DATA_BLOCK "DB_NcVarSelect_MA_POS_LIMIT_MINUS2"   // DB67
{ S7_Optimized_Access := 'TRUE' }
// stored: MemoryReserve 100
   VAR
      "$MA_POS_LIMIT_MINUS2_Axis01_X" { S7_SetPoint := 'True'} : "LBP_typeNCVariableTokenLReal";
      "$MA_POS_LIMIT_MINUS2_Axis02_Y" { S7_SetPoint := 'True'} : "LBP_typeNCVariableTokenLReal";
      "$MA_POS_LIMIT_MINUS2_Axis03_ZM" { S7_SetPoint := 'True'} : "LBP_typeNCVariableTokenLReal";
      "$MA_POS_LIMIT_MINUS2_Axis04_B" { S7_SetPoint := 'True'} : "LBP_typeNCVariableTokenLReal";
      "$MA_POS_LIMIT_MINUS2_Axis05_U1" { S7_SetPoint := 'True'} : "LBP_typeNCVariableTokenLReal";
      "$MA_POS_LIMIT_MINUS2_Axis06_U2" { S7_SetPoint := 'True'} : "LBP_typeNCVariableTokenLReal";
      "$MA_POS_LIMIT_MINUS2_Axis07_V" { S7_SetPoint := 'True'} : "LBP_typeNCVariableTokenLReal";
      "$MA_POS_LIMIT_MINUS2_Axis08_W" { S7_SetPoint := 'True'} : "LBP_typeNCVariableTokenLReal";
      "$MA_POS_LIMIT_MINUS2_Axis09_ZL" { S7_SetPoint := 'True'} : "LBP_typeNCVariableTokenLReal";
   END_VAR
BEGIN
   "$MA_POS_LIMIT_MINUS2_Axis01_X".token.syntaxId := 16#82;
   "$MA_POS_LIMIT_MINUS2_Axis01_X".token.areaAndUnit := 16#61;
   "$MA_POS_LIMIT_MINUS2_Axis01_X".token.column := 16#8D18;
   "$MA_POS_LIMIT_MINUS2_Axis01_X".token.row := 16#1;
   "$MA_POS_LIMIT_MINUS2_Axis01_X".token.blockType := 16#1A;
   "$MA_POS_LIMIT_MINUS2_Axis01_X".token.numberOfRows := 16#1;
   "$MA_POS_LIMIT_MINUS2_Axis01_X".token.dataTypeCode := 16#F;
   "$MA_POS_LIMIT_MINUS2_Axis01_X".token.length := 16#8;
   "$MA_POS_LIMIT_MINUS2_Axis02_Y".token.syntaxId := 16#82;
   "$MA_POS_LIMIT_MINUS2_Axis02_Y".token.areaAndUnit := 16#62;
   "$MA_POS_LIMIT_MINUS2_Axis02_Y".token.column := 16#8D18;
   "$MA_POS_LIMIT_MINUS2_Axis02_Y".token.row := 16#1;
   "$MA_POS_LIMIT_MINUS2_Axis02_Y".token.blockType := 16#1A;
   "$MA_POS_LIMIT_MINUS2_Axis02_Y".token.numberOfRows := 16#1;
   "$MA_POS_LIMIT_MINUS2_Axis02_Y".token.dataTypeCode := 16#F;
   "$MA_POS_LIMIT_MINUS2_Axis02_Y".token.length := 16#8;
   "$MA_POS_LIMIT_MINUS2_Axis03_ZM".token.syntaxId := 16#82;
   "$MA_POS_LIMIT_MINUS2_Axis03_ZM".token.areaAndUnit := 16#63;
   "$MA_POS_LIMIT_MINUS2_Axis03_ZM".token.column := 16#8D18;
   "$MA_POS_LIMIT_MINUS2_Axis03_ZM".token.row := 16#1;
   "$MA_POS_LIMIT_MINUS2_Axis03_ZM".token.blockType := 16#1A;
   "$MA_POS_LIMIT_MINUS2_Axis03_ZM".token.numberOfRows := 16#1;
   "$MA_POS_LIMIT_MINUS2_Axis03_ZM".token.dataTypeCode := 16#F;
   "$MA_POS_LIMIT_MINUS2_Axis03_ZM".token.length := 16#8;
   "$MA_POS_LIMIT_MINUS2_Axis04_B".token.syntaxId := 16#82;
   "$MA_POS_LIMIT_MINUS2_Axis04_B".token.areaAndUnit := 16#64;
   "$MA_POS_LIMIT_MINUS2_Axis04_B".token.column := 16#8D18;
   "$MA_POS_LIMIT_MINUS2_Axis04_B".token.row := 16#1;
   "$MA_POS_LIMIT_MINUS2_Axis04_B".token.blockType := 16#1A;
   "$MA_POS_LIMIT_MINUS2_Axis04_B".token.numberOfRows := 16#1;
   "$MA_POS_LIMIT_MINUS2_Axis04_B".token.dataTypeCode := 16#F;
   "$MA_POS_LIMIT_MINUS2_Axis04_B".token.length := 16#8;
   "$MA_POS_LIMIT_MINUS2_Axis05_U1".token.syntaxId := 16#82;
   "$MA_POS_LIMIT_MINUS2_Axis05_U1".token.areaAndUnit := 16#65;
   "$MA_POS_LIMIT_MINUS2_Axis05_U1".token.column := 16#8D18;
   "$MA_POS_LIMIT_MINUS2_Axis05_U1".token.row := 16#1;
   "$MA_POS_LIMIT_MINUS2_Axis05_U1".token.blockType := 16#1A;
   "$MA_POS_LIMIT_MINUS2_Axis05_U1".token.numberOfRows := 16#1;
   "$MA_POS_LIMIT_MINUS2_Axis05_U1".token.dataTypeCode := 16#F;
   "$MA_POS_LIMIT_MINUS2_Axis05_U1".token.length := 16#8;
   "$MA_POS_LIMIT_MINUS2_Axis06_U2".token.syntaxId := 16#82;
   "$MA_POS_LIMIT_MINUS2_Axis06_U2".token.areaAndUnit := 16#66;
   "$MA_POS_LIMIT_MINUS2_Axis06_U2".token.column := 16#8D18;
   "$MA_POS_LIMIT_MINUS2_Axis06_U2".token.row := 16#1;
   "$MA_POS_LIMIT_MINUS2_Axis06_U2".token.blockType := 16#1A;
   "$MA_POS_LIMIT_MINUS2_Axis06_U2".token.numberOfRows := 16#1;
   "$MA_POS_LIMIT_MINUS2_Axis06_U2".token.dataTypeCode := 16#F;
   "$MA_POS_LIMIT_MINUS2_Axis06_U2".token.length := 16#8;
   "$MA_POS_LIMIT_MINUS2_Axis07_V".token.syntaxId := 16#82;
   "$MA_POS_LIMIT_MINUS2_Axis07_V".token.areaAndUnit := 16#67;
   "$MA_POS_LIMIT_MINUS2_Axis07_V".token.column := 16#8D18;
   "$MA_POS_LIMIT_MINUS2_Axis07_V".token.row := 16#1;
   "$MA_POS_LIMIT_MINUS2_Axis07_V".token.blockType := 16#1A;
   "$MA_POS_LIMIT_MINUS2_Axis07_V".token.numberOfRows := 16#1;
   "$MA_POS_LIMIT_MINUS2_Axis07_V".token.dataTypeCode := 16#F;
   "$MA_POS_LIMIT_MINUS2_Axis07_V".token.length := 16#8;
   "$MA_POS_LIMIT_MINUS2_Axis08_W".token.syntaxId := 16#82;
   "$MA_POS_LIMIT_MINUS2_Axis08_W".token.areaAndUnit := 16#68;
   "$MA_POS_LIMIT_MINUS2_Axis08_W".token.column := 16#8D18;
   "$MA_POS_LIMIT_MINUS2_Axis08_W".token.row := 16#1;
   "$MA_POS_LIMIT_MINUS2_Axis08_W".token.blockType := 16#1A;
   "$MA_POS_LIMIT_MINUS2_Axis08_W".token.numberOfRows := 16#1;
   "$MA_POS_LIMIT_MINUS2_Axis08_W".token.dataTypeCode := 16#F;
   "$MA_POS_LIMIT_MINUS2_Axis08_W".token.length := 16#8;
   "$MA_POS_LIMIT_MINUS2_Axis09_ZL".token.syntaxId := 16#82;
   "$MA_POS_LIMIT_MINUS2_Axis09_ZL".token.areaAndUnit := 16#69;
   "$MA_POS_LIMIT_MINUS2_Axis09_ZL".token.column := 16#8D18;
   "$MA_POS_LIMIT_MINUS2_Axis09_ZL".token.row := 16#1;
   "$MA_POS_LIMIT_MINUS2_Axis09_ZL".token.blockType := 16#1A;
   "$MA_POS_LIMIT_MINUS2_Axis09_ZL".token.numberOfRows := 16#1;
   "$MA_POS_LIMIT_MINUS2_Axis09_ZL".token.dataTypeCode := 16#F;
   "$MA_POS_LIMIT_MINUS2_Axis09_ZL".token.length := 16#8;
END_DATA_BLOCK

DATA_BLOCK "DB_NcVarSelect_MA_POS_LIMIT_PLUS"   // DB68
{ S7_Optimized_Access := 'TRUE' }
// stored: MemoryReserve 100
   VAR
      "$MA_POS_LIMIT_PLUS_Axis01_X" { S7_SetPoint := 'True'} : SINU_typeNcVarTokenLReal;
      "$MA_POS_LIMIT_PLUS_Axis02_Y" { S7_SetPoint := 'True'} : SINU_typeNcVarTokenLReal;
      "$MA_POS_LIMIT_PLUS_Axis03_ZM" { S7_SetPoint := 'True'} : SINU_typeNcVarTokenLReal;
      "$MA_POS_LIMIT_PLUS_Axis04_B" { S7_SetPoint := 'True'} : SINU_typeNcVarTokenLReal;
      "$MA_POS_LIMIT_PLUS_Axis05_U1" { S7_SetPoint := 'True'} : SINU_typeNcVarTokenLReal;
      "$MA_POS_LIMIT_PLUS_Axis06_U2" { S7_SetPoint := 'True'} : SINU_typeNcVarTokenLReal;
      "$MA_POS_LIMIT_PLUS_Axis07_V" { S7_SetPoint := 'True'} : SINU_typeNcVarTokenLReal;
      "$MA_POS_LIMIT_PLUS_Axis08_W" { S7_SetPoint := 'True'} : SINU_typeNcVarTokenLReal;
      "$MA_POS_LIMIT_PLUS_Axis09_ZL" { S7_SetPoint := 'True'} : SINU_typeNcVarTokenLReal;
   END_VAR
BEGIN
   "$MA_POS_LIMIT_PLUS_Axis01_X".token.syntaxId := 16#82;
   "$MA_POS_LIMIT_PLUS_Axis01_X".token.areaAndUnit := 16#61;
   "$MA_POS_LIMIT_PLUS_Axis01_X".token.column := 16#8D0E;
   "$MA_POS_LIMIT_PLUS_Axis01_X".token.row := 16#1;
   "$MA_POS_LIMIT_PLUS_Axis01_X".token.blockType := 16#1A;
   "$MA_POS_LIMIT_PLUS_Axis01_X".token.rowCount := 16#1;
   "$MA_POS_LIMIT_PLUS_Axis01_X".token.dataType := 16#F;
   "$MA_POS_LIMIT_PLUS_Axis01_X".token.length := 16#8;
   "$MA_POS_LIMIT_PLUS_Axis02_Y".token.syntaxId := 16#82;
   "$MA_POS_LIMIT_PLUS_Axis02_Y".token.areaAndUnit := 16#62;
   "$MA_POS_LIMIT_PLUS_Axis02_Y".token.column := 16#8D0E;
   "$MA_POS_LIMIT_PLUS_Axis02_Y".token.row := 16#1;
   "$MA_POS_LIMIT_PLUS_Axis02_Y".token.blockType := 16#1A;
   "$MA_POS_LIMIT_PLUS_Axis02_Y".token.rowCount := 16#1;
   "$MA_POS_LIMIT_PLUS_Axis02_Y".token.dataType := 16#F;
   "$MA_POS_LIMIT_PLUS_Axis02_Y".token.length := 16#8;
   "$MA_POS_LIMIT_PLUS_Axis03_ZM".token.syntaxId := 16#82;
   "$MA_POS_LIMIT_PLUS_Axis03_ZM".token.areaAndUnit := 16#63;
   "$MA_POS_LIMIT_PLUS_Axis03_ZM".token.column := 16#8D0E;
   "$MA_POS_LIMIT_PLUS_Axis03_ZM".token.row := 16#1;
   "$MA_POS_LIMIT_PLUS_Axis03_ZM".token.blockType := 16#1A;
   "$MA_POS_LIMIT_PLUS_Axis03_ZM".token.rowCount := 16#1;
   "$MA_POS_LIMIT_PLUS_Axis03_ZM".token.dataType := 16#F;
   "$MA_POS_LIMIT_PLUS_Axis03_ZM".token.length := 16#8;
   "$MA_POS_LIMIT_PLUS_Axis04_B".token.syntaxId := 16#82;
   "$MA_POS_LIMIT_PLUS_Axis04_B".token.areaAndUnit := 16#64;
   "$MA_POS_LIMIT_PLUS_Axis04_B".token.column := 16#8D0E;
   "$MA_POS_LIMIT_PLUS_Axis04_B".token.row := 16#1;
   "$MA_POS_LIMIT_PLUS_Axis04_B".token.blockType := 16#1A;
   "$MA_POS_LIMIT_PLUS_Axis04_B".token.rowCount := 16#1;
   "$MA_POS_LIMIT_PLUS_Axis04_B".token.dataType := 16#F;
   "$MA_POS_LIMIT_PLUS_Axis04_B".token.length := 16#8;
   "$MA_POS_LIMIT_PLUS_Axis05_U1".token.syntaxId := 16#82;
   "$MA_POS_LIMIT_PLUS_Axis05_U1".token.areaAndUnit := 16#65;
   "$MA_POS_LIMIT_PLUS_Axis05_U1".token.column := 16#8D0E;
   "$MA_POS_LIMIT_PLUS_Axis05_U1".token.row := 16#1;
   "$MA_POS_LIMIT_PLUS_Axis05_U1".token.blockType := 16#1A;
   "$MA_POS_LIMIT_PLUS_Axis05_U1".token.rowCount := 16#1;
   "$MA_POS_LIMIT_PLUS_Axis05_U1".token.dataType := 16#F;
   "$MA_POS_LIMIT_PLUS_Axis05_U1".token.length := 16#8;
   "$MA_POS_LIMIT_PLUS_Axis06_U2".token.syntaxId := 16#82;
   "$MA_POS_LIMIT_PLUS_Axis06_U2".token.areaAndUnit := 16#66;
   "$MA_POS_LIMIT_PLUS_Axis06_U2".token.column := 16#8D0E;
   "$MA_POS_LIMIT_PLUS_Axis06_U2".token.row := 16#1;
   "$MA_POS_LIMIT_PLUS_Axis06_U2".token.blockType := 16#1A;
   "$MA_POS_LIMIT_PLUS_Axis06_U2".token.rowCount := 16#1;
   "$MA_POS_LIMIT_PLUS_Axis06_U2".token.dataType := 16#F;
   "$MA_POS_LIMIT_PLUS_Axis06_U2".token.length := 16#8;
   "$MA_POS_LIMIT_PLUS_Axis07_V".token.syntaxId := 16#82;
   "$MA_POS_LIMIT_PLUS_Axis07_V".token.areaAndUnit := 16#67;
   "$MA_POS_LIMIT_PLUS_Axis07_V".token.column := 16#8D0E;
   "$MA_POS_LIMIT_PLUS_Axis07_V".token.row := 16#1;
   "$MA_POS_LIMIT_PLUS_Axis07_V".token.blockType := 16#1A;
   "$MA_POS_LIMIT_PLUS_Axis07_V".token.rowCount := 16#1;
   "$MA_POS_LIMIT_PLUS_Axis07_V".token.dataType := 16#F;
   "$MA_POS_LIMIT_PLUS_Axis07_V".token.length := 16#8;
   "$MA_POS_LIMIT_PLUS_Axis08_W".token.syntaxId := 16#82;
   "$MA_POS_LIMIT_PLUS_Axis08_W".token.areaAndUnit := 16#68;
   "$MA_POS_LIMIT_PLUS_Axis08_W".token.column := 16#8D0E;
   "$MA_POS_LIMIT_PLUS_Axis08_W".token.row := 16#1;
   "$MA_POS_LIMIT_PLUS_Axis08_W".token.blockType := 16#1A;
   "$MA_POS_LIMIT_PLUS_Axis08_W".token.rowCount := 16#1;
   "$MA_POS_LIMIT_PLUS_Axis08_W".token.dataType := 16#F;
   "$MA_POS_LIMIT_PLUS_Axis08_W".token.length := 16#8;
   "$MA_POS_LIMIT_PLUS_Axis09_ZL".token.syntaxId := 16#82;
   "$MA_POS_LIMIT_PLUS_Axis09_ZL".token.areaAndUnit := 16#69;
   "$MA_POS_LIMIT_PLUS_Axis09_ZL".token.column := 16#8D0E;
   "$MA_POS_LIMIT_PLUS_Axis09_ZL".token.row := 16#1;
   "$MA_POS_LIMIT_PLUS_Axis09_ZL".token.blockType := 16#1A;
   "$MA_POS_LIMIT_PLUS_Axis09_ZL".token.rowCount := 16#1;
   "$MA_POS_LIMIT_PLUS_Axis09_ZL".token.dataType := 16#F;
   "$MA_POS_LIMIT_PLUS_Axis09_ZL".token.length := 16#8;
END_DATA_BLOCK

DATA_BLOCK "DB_NcVarSelect_MA_POS_LIMIT_PLUS2"   // DB69
{ S7_Optimized_Access := 'TRUE' }
// stored: MemoryReserve 100
   VAR
      "$MA_POS_LIMIT_PLUS2_Axis01_X" { S7_SetPoint := 'True'} : "LBP_typeNCVariableTokenLReal";
      "$MA_POS_LIMIT_PLUS2_Axis02_Y" { S7_SetPoint := 'True'} : "LBP_typeNCVariableTokenLReal";
      "$MA_POS_LIMIT_PLUS2_Axis03_ZM" { S7_SetPoint := 'True'} : "LBP_typeNCVariableTokenLReal";
      "$MA_POS_LIMIT_PLUS2_Axis04_B" { S7_SetPoint := 'True'} : "LBP_typeNCVariableTokenLReal";
      "$MA_POS_LIMIT_PLUS2_Axis05_U1" { S7_SetPoint := 'True'} : "LBP_typeNCVariableTokenLReal";
      "$MA_POS_LIMIT_PLUS2_Axis06_U2" { S7_SetPoint := 'True'} : "LBP_typeNCVariableTokenLReal";
      "$MA_POS_LIMIT_PLUS2_Axis07_V" { S7_SetPoint := 'True'} : "LBP_typeNCVariableTokenLReal";
      "$MA_POS_LIMIT_PLUS2_Axis08_W" { S7_SetPoint := 'True'} : "LBP_typeNCVariableTokenLReal";
      "$MA_POS_LIMIT_PLUS2_Axis09_ZL" { S7_SetPoint := 'True'} : "LBP_typeNCVariableTokenLReal";
   END_VAR
BEGIN
   "$MA_POS_LIMIT_PLUS2_Axis01_X".token.syntaxId := 16#82;
   "$MA_POS_LIMIT_PLUS2_Axis01_X".token.areaAndUnit := 16#61;
   "$MA_POS_LIMIT_PLUS2_Axis01_X".token.column := 16#8D22;
   "$MA_POS_LIMIT_PLUS2_Axis01_X".token.row := 16#1;
   "$MA_POS_LIMIT_PLUS2_Axis01_X".token.blockType := 16#1A;
   "$MA_POS_LIMIT_PLUS2_Axis01_X".token.numberOfRows := 16#1;
   "$MA_POS_LIMIT_PLUS2_Axis01_X".token.dataTypeCode := 16#F;
   "$MA_POS_LIMIT_PLUS2_Axis01_X".token.length := 16#8;
   "$MA_POS_LIMIT_PLUS2_Axis02_Y".token.syntaxId := 16#82;
   "$MA_POS_LIMIT_PLUS2_Axis02_Y".token.areaAndUnit := 16#62;
   "$MA_POS_LIMIT_PLUS2_Axis02_Y".token.column := 16#8D22;
   "$MA_POS_LIMIT_PLUS2_Axis02_Y".token.row := 16#1;
   "$MA_POS_LIMIT_PLUS2_Axis02_Y".token.blockType := 16#1A;
   "$MA_POS_LIMIT_PLUS2_Axis02_Y".token.numberOfRows := 16#1;
   "$MA_POS_LIMIT_PLUS2_Axis02_Y".token.dataTypeCode := 16#F;
   "$MA_POS_LIMIT_PLUS2_Axis02_Y".token.length := 16#8;
   "$MA_POS_LIMIT_PLUS2_Axis03_ZM".token.syntaxId := 16#82;
   "$MA_POS_LIMIT_PLUS2_Axis03_ZM".token.areaAndUnit := 16#63;
   "$MA_POS_LIMIT_PLUS2_Axis03_ZM".token.column := 16#8D22;
   "$MA_POS_LIMIT_PLUS2_Axis03_ZM".token.row := 16#1;
   "$MA_POS_LIMIT_PLUS2_Axis03_ZM".token.blockType := 16#1A;
   "$MA_POS_LIMIT_PLUS2_Axis03_ZM".token.numberOfRows := 16#1;
   "$MA_POS_LIMIT_PLUS2_Axis03_ZM".token.dataTypeCode := 16#F;
   "$MA_POS_LIMIT_PLUS2_Axis03_ZM".token.length := 16#8;
   "$MA_POS_LIMIT_PLUS2_Axis04_B".token.syntaxId := 16#82;
   "$MA_POS_LIMIT_PLUS2_Axis04_B".token.areaAndUnit := 16#64;
   "$MA_POS_LIMIT_PLUS2_Axis04_B".token.column := 16#8D22;
   "$MA_POS_LIMIT_PLUS2_Axis04_B".token.row := 16#1;
   "$MA_POS_LIMIT_PLUS2_Axis04_B".token.blockType := 16#1A;
   "$MA_POS_LIMIT_PLUS2_Axis04_B".token.numberOfRows := 16#1;
   "$MA_POS_LIMIT_PLUS2_Axis04_B".token.dataTypeCode := 16#F;
   "$MA_POS_LIMIT_PLUS2_Axis04_B".token.length := 16#8;
   "$MA_POS_LIMIT_PLUS2_Axis05_U1".token.syntaxId := 16#82;
   "$MA_POS_LIMIT_PLUS2_Axis05_U1".token.areaAndUnit := 16#65;
   "$MA_POS_LIMIT_PLUS2_Axis05_U1".token.column := 16#8D22;
   "$MA_POS_LIMIT_PLUS2_Axis05_U1".token.row := 16#1;
   "$MA_POS_LIMIT_PLUS2_Axis05_U1".token.blockType := 16#1A;
   "$MA_POS_LIMIT_PLUS2_Axis05_U1".token.numberOfRows := 16#1;
   "$MA_POS_LIMIT_PLUS2_Axis05_U1".token.dataTypeCode := 16#F;
   "$MA_POS_LIMIT_PLUS2_Axis05_U1".token.length := 16#8;
   "$MA_POS_LIMIT_PLUS2_Axis06_U2".token.syntaxId := 16#82;
   "$MA_POS_LIMIT_PLUS2_Axis06_U2".token.areaAndUnit := 16#66;
   "$MA_POS_LIMIT_PLUS2_Axis06_U2".token.column := 16#8D22;
   "$MA_POS_LIMIT_PLUS2_Axis06_U2".token.row := 16#1;
   "$MA_POS_LIMIT_PLUS2_Axis06_U2".token.blockType := 16#1A;
   "$MA_POS_LIMIT_PLUS2_Axis06_U2".token.numberOfRows := 16#1;
   "$MA_POS_LIMIT_PLUS2_Axis06_U2".token.dataTypeCode := 16#F;
   "$MA_POS_LIMIT_PLUS2_Axis06_U2".token.length := 16#8;
   "$MA_POS_LIMIT_PLUS2_Axis07_V".token.syntaxId := 16#82;
   "$MA_POS_LIMIT_PLUS2_Axis07_V".token.areaAndUnit := 16#67;
   "$MA_POS_LIMIT_PLUS2_Axis07_V".token.column := 16#8D22;
   "$MA_POS_LIMIT_PLUS2_Axis07_V".token.row := 16#1;
   "$MA_POS_LIMIT_PLUS2_Axis07_V".token.blockType := 16#1A;
   "$MA_POS_LIMIT_PLUS2_Axis07_V".token.numberOfRows := 16#1;
   "$MA_POS_LIMIT_PLUS2_Axis07_V".token.dataTypeCode := 16#F;
   "$MA_POS_LIMIT_PLUS2_Axis07_V".token.length := 16#8;
   "$MA_POS_LIMIT_PLUS2_Axis08_W".token.syntaxId := 16#82;
   "$MA_POS_LIMIT_PLUS2_Axis08_W".token.areaAndUnit := 16#68;
   "$MA_POS_LIMIT_PLUS2_Axis08_W".token.column := 16#8D22;
   "$MA_POS_LIMIT_PLUS2_Axis08_W".token.row := 16#1;
   "$MA_POS_LIMIT_PLUS2_Axis08_W".token.blockType := 16#1A;
   "$MA_POS_LIMIT_PLUS2_Axis08_W".token.numberOfRows := 16#1;
   "$MA_POS_LIMIT_PLUS2_Axis08_W".token.dataTypeCode := 16#F;
   "$MA_POS_LIMIT_PLUS2_Axis08_W".token.length := 16#8;
   "$MA_POS_LIMIT_PLUS2_Axis09_ZL".token.syntaxId := 16#82;
   "$MA_POS_LIMIT_PLUS2_Axis09_ZL".token.areaAndUnit := 16#69;
   "$MA_POS_LIMIT_PLUS2_Axis09_ZL".token.column := 16#8D22;
   "$MA_POS_LIMIT_PLUS2_Axis09_ZL".token.row := 16#1;
   "$MA_POS_LIMIT_PLUS2_Axis09_ZL".token.blockType := 16#1A;
   "$MA_POS_LIMIT_PLUS2_Axis09_ZL".token.numberOfRows := 16#1;
   "$MA_POS_LIMIT_PLUS2_Axis09_ZL".token.dataTypeCode := 16#F;
   "$MA_POS_LIMIT_PLUS2_Axis09_ZL".token.length := 16#8;
END_DATA_BLOCK

DATA_BLOCK "DB_NcVarSelect_M_MAX_AX_VELO"   // DB98
{ S7_Optimized_Access := 'TRUE' }
// stored: MemoryReserve 100
   VAR
      "$MA_JOG_VELO_Axis01_X" { S7_SetPoint := 'True'} : "LBP_typeNCVariableTokenLReal";
      "$MA_JOG_VELO_Axis02_Y" { S7_SetPoint := 'True'} : "LBP_typeNCVariableTokenLReal";
      "$MA_JOG_VELO_Axis03_ZM" { S7_SetPoint := 'True'} : "LBP_typeNCVariableTokenLReal";
      "$MA_JOG_VELO_Axis04_B" { S7_SetPoint := 'True'} : "LBP_typeNCVariableTokenLReal";
      "$MA_JOG_VELO_Axis05_U1" { S7_SetPoint := 'True'} : "LBP_typeNCVariableTokenLReal";
      "$MA_JOG_VELO_Axis06_U2" { S7_SetPoint := 'True'} : "LBP_typeNCVariableTokenLReal";
      "$MA_JOG_VELO_Axis07_V" { S7_SetPoint := 'True'} : "LBP_typeNCVariableTokenLReal";
      "$MA_JOG_VELO_Axis08_W" { S7_SetPoint := 'True'} : "LBP_typeNCVariableTokenLReal";
      "$MA_JOG_VELO_Axis09_ZL" { S7_SetPoint := 'True'} : "LBP_typeNCVariableTokenLReal";
   END_VAR
BEGIN
   "$MA_JOG_VELO_Axis01_X".token.syntaxId := 16#82;
   "$MA_JOG_VELO_Axis01_X".token.areaAndUnit := 16#61;
   "$MA_JOG_VELO_Axis01_X".token.column := 16#7D00;
   "$MA_JOG_VELO_Axis01_X".token.row := 16#1;
   "$MA_JOG_VELO_Axis01_X".token.blockType := 16#1A;
   "$MA_JOG_VELO_Axis01_X".token.numberOfRows := 16#1;
   "$MA_JOG_VELO_Axis01_X".token.dataTypeCode := 16#F;
   "$MA_JOG_VELO_Axis01_X".token.length := 16#8;
   "$MA_JOG_VELO_Axis02_Y".token.syntaxId := 16#82;
   "$MA_JOG_VELO_Axis02_Y".token.areaAndUnit := 16#62;
   "$MA_JOG_VELO_Axis02_Y".token.column := 16#7D00;
   "$MA_JOG_VELO_Axis02_Y".token.row := 16#1;
   "$MA_JOG_VELO_Axis02_Y".token.blockType := 16#1A;
   "$MA_JOG_VELO_Axis02_Y".token.numberOfRows := 16#1;
   "$MA_JOG_VELO_Axis02_Y".token.dataTypeCode := 16#F;
   "$MA_JOG_VELO_Axis02_Y".token.length := 16#8;
   "$MA_JOG_VELO_Axis03_ZM".token.syntaxId := 16#82;
   "$MA_JOG_VELO_Axis03_ZM".token.areaAndUnit := 16#63;
   "$MA_JOG_VELO_Axis03_ZM".token.column := 16#7D00;
   "$MA_JOG_VELO_Axis03_ZM".token.row := 16#1;
   "$MA_JOG_VELO_Axis03_ZM".token.blockType := 16#1A;
   "$MA_JOG_VELO_Axis03_ZM".token.numberOfRows := 16#1;
   "$MA_JOG_VELO_Axis03_ZM".token.dataTypeCode := 16#F;
   "$MA_JOG_VELO_Axis03_ZM".token.length := 16#8;
   "$MA_JOG_VELO_Axis04_B".token.syntaxId := 16#82;
   "$MA_JOG_VELO_Axis04_B".token.areaAndUnit := 16#64;
   "$MA_JOG_VELO_Axis04_B".token.column := 16#7D00;
   "$MA_JOG_VELO_Axis04_B".token.row := 16#1;
   "$MA_JOG_VELO_Axis04_B".token.blockType := 16#1A;
   "$MA_JOG_VELO_Axis04_B".token.numberOfRows := 16#1;
   "$MA_JOG_VELO_Axis04_B".token.dataTypeCode := 16#F;
   "$MA_JOG_VELO_Axis04_B".token.length := 16#8;
   "$MA_JOG_VELO_Axis05_U1".token.syntaxId := 16#82;
   "$MA_JOG_VELO_Axis05_U1".token.areaAndUnit := 16#65;
   "$MA_JOG_VELO_Axis05_U1".token.column := 16#7D00;
   "$MA_JOG_VELO_Axis05_U1".token.row := 16#1;
   "$MA_JOG_VELO_Axis05_U1".token.blockType := 16#1A;
   "$MA_JOG_VELO_Axis05_U1".token.numberOfRows := 16#1;
   "$MA_JOG_VELO_Axis05_U1".token.dataTypeCode := 16#F;
   "$MA_JOG_VELO_Axis05_U1".token.length := 16#8;
   "$MA_JOG_VELO_Axis06_U2".token.syntaxId := 16#82;
   "$MA_JOG_VELO_Axis06_U2".token.areaAndUnit := 16#66;
   "$MA_JOG_VELO_Axis06_U2".token.column := 16#7D00;
   "$MA_JOG_VELO_Axis06_U2".token.row := 16#1;
   "$MA_JOG_VELO_Axis06_U2".token.blockType := 16#1A;
   "$MA_JOG_VELO_Axis06_U2".token.numberOfRows := 16#1;
   "$MA_JOG_VELO_Axis06_U2".token.dataTypeCode := 16#F;
   "$MA_JOG_VELO_Axis06_U2".token.length := 16#8;
   "$MA_JOG_VELO_Axis07_V".token.syntaxId := 16#82;
   "$MA_JOG_VELO_Axis07_V".token.areaAndUnit := 16#67;
   "$MA_JOG_VELO_Axis07_V".token.column := 16#7D00;
   "$MA_JOG_VELO_Axis07_V".token.row := 16#1;
   "$MA_JOG_VELO_Axis07_V".token.blockType := 16#1A;
   "$MA_JOG_VELO_Axis07_V".token.numberOfRows := 16#1;
   "$MA_JOG_VELO_Axis07_V".token.dataTypeCode := 16#F;
   "$MA_JOG_VELO_Axis07_V".token.length := 16#8;
   "$MA_JOG_VELO_Axis08_W".token.syntaxId := 16#82;
   "$MA_JOG_VELO_Axis08_W".token.areaAndUnit := 16#68;
   "$MA_JOG_VELO_Axis08_W".token.column := 16#7D00;
   "$MA_JOG_VELO_Axis08_W".token.row := 16#1;
   "$MA_JOG_VELO_Axis08_W".token.blockType := 16#1A;
   "$MA_JOG_VELO_Axis08_W".token.numberOfRows := 16#1;
   "$MA_JOG_VELO_Axis08_W".token.dataTypeCode := 16#F;
   "$MA_JOG_VELO_Axis08_W".token.length := 16#8;
   "$MA_JOG_VELO_Axis09_ZL".token.syntaxId := 16#82;
   "$MA_JOG_VELO_Axis09_ZL".token.areaAndUnit := 16#69;
   "$MA_JOG_VELO_Axis09_ZL".token.column := 16#7D00;
   "$MA_JOG_VELO_Axis09_ZL".token.row := 16#1;
   "$MA_JOG_VELO_Axis09_ZL".token.blockType := 16#1A;
   "$MA_JOG_VELO_Axis09_ZL".token.numberOfRows := 16#1;
   "$MA_JOG_VELO_Axis09_ZL".token.dataTypeCode := 16#F;
   "$MA_JOG_VELO_Axis09_ZL".token.length := 16#8;
END_DATA_BLOCK

DATA_BLOCK "DB_AnalogInputAction"   // DB1304
TITLE = TEMPERATURE SETTINGS
{ S7_Optimized_Access := 'FALSE'; DB_Accessible_From_OPC_UA := 'FALSE' }
AUTHOR : SAN
// stored: AutoNumber false, DBAccessibleFromOPCUA false, DBAccessibleFromWebserver false
   VAR
      Laser_Power_Meter : "AnalogInAction_DT";
      Axis_B_Clamping_Part : "AnalogInAction_DT";
      Laser_Air_Pressure_Process : "AnalogInAction_DT";
      Inlet_Air_Pressure : "AnalogInAction_DT";
      Ambiant_Temperature : "AnalogInAction_DT";
      Machine_Temperature : "AnalogInAction_DT";
      Cold_Water_Temperature_Input : "AnalogInAction_DT";
      Cold_Water_Temperature_Output : "AnalogInAction_DT";
      X_Axis_Temperature_PT1000 : "AnalogInAction_DT";
      Y_Axis_Temperature_PT1000 : "AnalogInAction_DT";
      X_Axis_Temperature_PTC : "AnalogInAction_DT";
      Y_Axis_Temperature_PTC : "AnalogInAction_DT";
      Nozzle_Overpressure : "AnalogInAction_DT";
      Optical_Path_Overpressure : "AnalogInAction_DT";
      Laser_Head_Overpressure : "AnalogInAction_DT";
      ZL_Axis_Overpressure : "AnalogInAction_DT";
      XY_Axis_Overpressure : "AnalogInAction_DT";
      Left_Aspiration : "AnalogInAction_DT";
      Right_Aspiration : "AnalogInAction_DT";
      Free_IW458 : "AnalogInAction_DT";
      Clim_Temperature : "AnalogInAction_DT";
      Free_IW482 : "AnalogInAction_DT";
      Free_IW484 : "AnalogInAction_DT";
      Free_IW486 : "AnalogInAction_DT";
      Sensor_Controller_Station1 : "AnalogInAction_DT";
      Cabinet_Temperature : "AnalogInAction_DT";
      Free_IW464 : "AnalogInAction_DT";
      Free_IW466 : "AnalogInAction_DT";
   END_VAR
BEGIN
   Laser_Power_Meter.ID_Measure := 1;
   Axis_B_Clamping_Part.ID_Measure := 2;
   Laser_Air_Pressure_Process.ID_Measure := 3;
   Inlet_Air_Pressure.ID_Measure := 4;
   Ambiant_Temperature.ID_Measure := 5;
   Machine_Temperature.ID_Measure := 6;
   Cold_Water_Temperature_Input.ID_Measure := 7;
   Cold_Water_Temperature_Output.ID_Measure := 8;
   X_Axis_Temperature_PT1000.ID_Measure := 9;
   Y_Axis_Temperature_PT1000.ID_Measure := 10;
   X_Axis_Temperature_PTC.ID_Measure := 11;
   Y_Axis_Temperature_PTC.ID_Measure := 12;
   Nozzle_Overpressure.ID_Measure := 13;
   Optical_Path_Overpressure.ID_Measure := 14;
   Laser_Head_Overpressure.ID_Measure := 15;
   ZL_Axis_Overpressure.ID_Measure := 16;
   XY_Axis_Overpressure.ID_Measure := 17;
   Left_Aspiration.ID_Measure := 18;
   Right_Aspiration.ID_Measure := 19;
   Free_IW458.ID_Measure := 20;
   Clim_Temperature.ID_Measure := 21;
   Free_IW482.ID_Measure := 22;
   Free_IW484.ID_Measure := 23;
   Free_IW486.ID_Measure := 24;
   Sensor_Controller_Station1.ID_Measure := 25;
   Cabinet_Temperature.ID_Measure := 26;
   Free_IW464.ID_Measure := 27;
   Free_IW466.ID_Measure := 28;
END_DATA_BLOCK

DATA_BLOCK "DB_AnalogInputDataHMI"   // DB1303
TITLE = TEMPERATURE SETTINGS
{ S7_Optimized_Access := 'FALSE'; DB_Accessible_From_OPC_UA := 'FALSE' }
AUTHOR : SAN
// stored: AutoNumber false, DBAccessibleFromOPCUA false, DBAccessibleFromWebserver false
   VAR RETAIN
      Laser_Power_Meter : "AnalogInDataHMI_DT";
      Axis_B_Clamping_Part : "AnalogInDataHMI_DT";
      Laser_Air_Pressure_Process : "AnalogInDataHMI_DT";
      Inlet_Air_Pressure : "AnalogInDataHMI_DT";
      Ambiant_Temperature : "AnalogInDataHMI_DT";
      Machine_Temperature : "AnalogInDataHMI_DT";
      Cold_Water_Temperature_Input : "AnalogInDataHMI_DT";
      Cold_Water_Temperature_Output : "AnalogInDataHMI_DT";
      X_Axis_Temperature_PT1000 { S7_SetPoint := 'True'} : "AnalogInDataHMI_DT";
      Y_Axis_Temperature_PT1000 : "AnalogInDataHMI_DT";
      X_Axis_Temperature_PTC : "AnalogInDataHMI_DT";
      Y_Axis_Temperature_PTC : "AnalogInDataHMI_DT";
      Nozzle_Overpressure : "AnalogInDataHMI_DT";
      Optical_Path_Overpressure : "AnalogInDataHMI_DT";
      Laser_Head_Overpressure : "AnalogInDataHMI_DT";
      ZL_Axis_Overpressure : "AnalogInDataHMI_DT";
      XY_Axis_Overpressure : "AnalogInDataHMI_DT";
      Left_Aspiration : "AnalogInDataHMI_DT";
      Right_Aspiration : "AnalogInDataHMI_DT";
      Free_IW458 : "AnalogInDataHMI_DT";
      Clim_Temperature : "AnalogInDataHMI_DT";
      Free_IW482 : "AnalogInDataHMI_DT";
      Free_IW484 : "AnalogInDataHMI_DT";
      Free_IW486 : "AnalogInDataHMI_DT";
      Sensor_Controller_Station1 : "AnalogInDataHMI_DT";
      Cabinet_Temperature : "AnalogInDataHMI_DT";
      Free_IW464 : "AnalogInDataHMI_DT";
      Free_IW466 : "AnalogInDataHMI_DT";
   END_VAR
BEGIN
   Laser_Power_Meter.ID_Measure := 701;
   Axis_B_Clamping_Part.ID_Measure := 810;
   Laser_Air_Pressure_Process.ID_Measure := 511;
   Laser_Air_Pressure_Process.TargetValue := 2.0;
   Laser_Air_Pressure_Process.ThresholdAlarmMin := -0.2;
   Laser_Air_Pressure_Process.ThresholdWarningMin := -0.15;
   Laser_Air_Pressure_Process.ThresholdWarningMax := 0.15;
   Laser_Air_Pressure_Process.ThresholdAlarmMax := 0.2;
   Laser_Air_Pressure_Process.StartTime := T#5s;
   Inlet_Air_Pressure.ID_Measure := 501;
   Inlet_Air_Pressure.TargetValue := 6.0;
   Inlet_Air_Pressure.ThresholdAlarmMin := -0.5;
   Inlet_Air_Pressure.ThresholdWarningMin := -0.4;
   Inlet_Air_Pressure.ThresholdWarningMax := 0.4;
   Inlet_Air_Pressure.ThresholdAlarmMax := 0.5;
   Inlet_Air_Pressure.StartTime := T#5s;
   Ambiant_Temperature.ID_Measure := 201;
   Ambiant_Temperature.TargetValue := 25.0;
   Ambiant_Temperature.ThresholdAlarmMin := -5.0;
   Ambiant_Temperature.ThresholdWarningMin := -3.0;
   Ambiant_Temperature.ThresholdWarningMax := 3.0;
   Ambiant_Temperature.ThresholdAlarmMax := 5.0;
   Machine_Temperature.ID_Measure := 202;
   Machine_Temperature.TargetValue := 25.0;
   Machine_Temperature.ThresholdAlarmMin := -5.0;
   Machine_Temperature.ThresholdWarningMin := -3.0;
   Machine_Temperature.ThresholdWarningMax := 3.0;
   Machine_Temperature.ThresholdAlarmMax := 5.0;
   Cold_Water_Temperature_Input.ID_Measure := 301;
   Cold_Water_Temperature_Input.TargetValue := 23.0;
   Cold_Water_Temperature_Input.ThresholdAlarmMin := -3.0;
   Cold_Water_Temperature_Input.ThresholdWarningMin := -2.0;
   Cold_Water_Temperature_Input.ThresholdWarningMax := 2.0;
   Cold_Water_Temperature_Input.ThresholdAlarmMax := 3.0;
   Cold_Water_Temperature_Output.ID_Measure := 302;
   Cold_Water_Temperature_Output.TargetValue := 24.0;
   Cold_Water_Temperature_Output.ThresholdAlarmMin := -3.0;
   Cold_Water_Temperature_Output.ThresholdWarningMin := -2.0;
   Cold_Water_Temperature_Output.ThresholdWarningMax := 2.0;
   Cold_Water_Temperature_Output.ThresholdAlarmMax := 3.0;
   X_Axis_Temperature_PT1000.ID_Measure := 110;
   X_Axis_Temperature_PT1000.TargetValue := 25.0;
   X_Axis_Temperature_PT1000.ThresholdAlarmMin := -5.0;
   X_Axis_Temperature_PT1000.ThresholdWarningMin := -3.0;
   X_Axis_Temperature_PT1000.ThresholdWarningMax := 3.0;
   X_Axis_Temperature_PT1000.ThresholdAlarmMax := 5.0;
   X_Axis_Temperature_PT1000.AxFactor := 1.0;
   X_Axis_Temperature_PT1000.StartTime := T#45S;
   Y_Axis_Temperature_PT1000.ID_Measure := 120;
   Y_Axis_Temperature_PT1000.TargetValue := 25.0;
   Y_Axis_Temperature_PT1000.ThresholdAlarmMin := -5.0;
   Y_Axis_Temperature_PT1000.ThresholdWarningMin := -3.0;
   Y_Axis_Temperature_PT1000.ThresholdWarningMax := 3.0;
   Y_Axis_Temperature_PT1000.ThresholdAlarmMax := 5.0;
   X_Axis_Temperature_PTC.ID_Measure := 116;
   Y_Axis_Temperature_PTC.ID_Measure := 126;
   Nozzle_Overpressure.ID_Measure := 512;
   Nozzle_Overpressure.TargetValue := 2.0;
   Nozzle_Overpressure.ThresholdAlarmMin := -0.2;
   Nozzle_Overpressure.ThresholdWarningMin := -0.15;
   Nozzle_Overpressure.ThresholdWarningMax := 0.15;
   Nozzle_Overpressure.ThresholdAlarmMax := 0.2;
   Nozzle_Overpressure.StartTime := T#5s;
   Optical_Path_Overpressure.ID_Measure := 513;
   Optical_Path_Overpressure.TargetValue := 0.4;
   Optical_Path_Overpressure.ThresholdAlarmMin := -0.2;
   Optical_Path_Overpressure.ThresholdWarningMin := -0.19;
   Optical_Path_Overpressure.ThresholdWarningMax := 0.19;
   Optical_Path_Overpressure.ThresholdAlarmMax := 0.2;
   Optical_Path_Overpressure.StartTime := T#5s;
   Laser_Head_Overpressure.ID_Measure := 514;
   Laser_Head_Overpressure.TargetValue := 1.4;
   Laser_Head_Overpressure.ThresholdAlarmMin := -0.15;
   Laser_Head_Overpressure.ThresholdWarningMin := -0.1;
   Laser_Head_Overpressure.ThresholdWarningMax := 0.1;
   Laser_Head_Overpressure.ThresholdAlarmMax := 0.15;
   Laser_Head_Overpressure.StartTime := T#5s;
   ZL_Axis_Overpressure.ID_Measure := 520;
   ZL_Axis_Overpressure.TargetValue := 0.85;
   ZL_Axis_Overpressure.ThresholdAlarmMin := -0.2;
   ZL_Axis_Overpressure.ThresholdWarningMin := -0.15;
   ZL_Axis_Overpressure.ThresholdWarningMax := 0.15;
   ZL_Axis_Overpressure.ThresholdAlarmMax := 0.2;
   ZL_Axis_Overpressure.StartTime := T#5s;
   XY_Axis_Overpressure.ID_Measure := 530;
   XY_Axis_Overpressure.TargetValue := 0.85;
   XY_Axis_Overpressure.ThresholdAlarmMin := -0.2;
   XY_Axis_Overpressure.ThresholdWarningMin := -0.15;
   XY_Axis_Overpressure.ThresholdWarningMax := 0.15;
   XY_Axis_Overpressure.ThresholdAlarmMax := 0.2;
   XY_Axis_Overpressure.StartTime := T#5s;
   Left_Aspiration.ID_Measure := 401;
   Left_Aspiration.CurrentValue := 1.4774;
   Left_Aspiration.TargetValue := 1900.0;
   Left_Aspiration.ThresholdAlarmMin := -1000.0;
   Left_Aspiration.ThresholdWarningMin := -500.0;
   Left_Aspiration.ThresholdWarningMax := 500.0;
   Left_Aspiration.ThresholdAlarmMax := 1000.0;
   Left_Aspiration.StartTime := T#120s;
   Right_Aspiration.ID_Measure := 402;
   Right_Aspiration.CurrentValue := 1.4774;
   Right_Aspiration.TargetValue := 1900.0;
   Right_Aspiration.ThresholdAlarmMin := -1000.0;
   Right_Aspiration.ThresholdWarningMin := -500.0;
   Right_Aspiration.ThresholdWarningMax := 500.0;
   Right_Aspiration.ThresholdAlarmMax := 1000.0;
   Right_Aspiration.StartTime := T#120s;
   Free_IW458.ID_Measure := 999;
   Clim_Temperature.ID_Measure := 204;
   Free_IW482.ID_Measure := 999;
   Free_IW484.ID_Measure := 999;
   Free_IW486.ID_Measure := 999;
   Sensor_Controller_Station1.ID_Measure := 711;
   Cabinet_Temperature.ID_Measure := 203;
   Free_IW464.ID_Measure := 999;
   Free_IW466.ID_Measure := 999;
END_DATA_BLOCK

DATA_BLOCK "DB_AnalogInputDataPLC"   // DB1307
TITLE = TEMPERATURE SETTINGS
{ S7_Optimized_Access := 'FALSE'; DB_Accessible_From_OPC_UA := 'FALSE' }
AUTHOR : SAN
// stored: AutoNumber false, DBAccessibleFromOPCUA false, DBAccessibleFromWebserver false
   VAR RETAIN
      Laser_Power_Meter : "AnalogInDataPLC_DT";
      Axis_B_Clamping_Part : "AnalogInDataPLC_DT";
      Laser_Air_Pressure_Process : "AnalogInDataPLC_DT";
      Inlet_Air_Pressure : "AnalogInDataPLC_DT";
      Ambiant_Temperature : "AnalogInDataPLC_DT";
      Machine_Temperature : "AnalogInDataPLC_DT";
      Cold_Water_Temperature_Input : "AnalogInDataPLC_DT";
      Cold_Water_Temperature_Output : "AnalogInDataPLC_DT";
      X_Axis_Temperature_PT1000 : "AnalogInDataPLC_DT";
      Y_Axis_Temperature_PT1000 : "AnalogInDataPLC_DT";
      X_Axis_Temperature_PTC : "AnalogInDataPLC_DT";
      Y_Axis_Temperature_PTC : "AnalogInDataPLC_DT";
      Nozzle_Overpressure : "AnalogInDataPLC_DT";
      Optical_Path_Overpressure : "AnalogInDataPLC_DT";
      Laser_Head_Overpressure : "AnalogInDataPLC_DT";
      ZL_Axis_Overpressure : "AnalogInDataPLC_DT";
      XY_Axis_Overpressure : "AnalogInDataPLC_DT";
      Left_Aspiration : "AnalogInDataPLC_DT";
      Right_Aspiration : "AnalogInDataPLC_DT";
      Free_IW458 : "AnalogInDataPLC_DT";
      Clim_Temperature : "AnalogInDataPLC_DT";
      Free_IW482 : "AnalogInDataPLC_DT";
      Free_IW484 : "AnalogInDataPLC_DT";
      Free_IW486 : "AnalogInDataPLC_DT";
      Sensor_Controller_Station1 : "AnalogInDataPLC_DT";
      Cabinet_Temperature : "AnalogInDataPLC_DT";
      Free_IW464 : "AnalogInDataPLC_DT";
      Free_IW466 : "AnalogInDataPLC_DT";
   END_VAR
BEGIN
   Laser_Power_Meter.LimitUp := 10.0;
   Laser_Power_Meter.LimitDown := 0.0;
   Laser_Power_Meter.TypeProbe := 2;
   Axis_B_Clamping_Part.LimitUp := 27648.0;
   Axis_B_Clamping_Part.LimitDown := 0.0;
   Axis_B_Clamping_Part.TypeProbe := 2;
   Laser_Air_Pressure_Process.LimitUp := 10.0;
   Laser_Air_Pressure_Process.LimitDown := 0.0;
   Laser_Air_Pressure_Process.TypeProbe := 2;
   Laser_Air_Pressure_Process.EnableAlarmMin := True;
   Laser_Air_Pressure_Process.EnableWarningMin := True;
   Laser_Air_Pressure_Process.EnableWarningMax := True;
   Laser_Air_Pressure_Process.EnableAlarmMax := True;
   Inlet_Air_Pressure.LimitUp := 10.0;
   Inlet_Air_Pressure.LimitDown := 0.0;
   Inlet_Air_Pressure.TypeProbe := 2;
   Inlet_Air_Pressure.EnableAlarmMin := True;
   Inlet_Air_Pressure.EnableWarningMin := True;
   Inlet_Air_Pressure.EnableWarningMax := True;
   Inlet_Air_Pressure.EnableAlarmMax := True;
   Ambiant_Temperature.TypeProbe := 0;
   Ambiant_Temperature.EnableAlarmMin := True;
   Ambiant_Temperature.EnableWarningMin := True;
   Ambiant_Temperature.EnableWarningMax := True;
   Ambiant_Temperature.EnableAlarmMax := True;
   Machine_Temperature.TypeProbe := 0;
   Machine_Temperature.EnableAlarmMin := True;
   Machine_Temperature.EnableWarningMin := True;
   Machine_Temperature.EnableWarningMax := True;
   Machine_Temperature.EnableAlarmMax := True;
   Cold_Water_Temperature_Input.TypeProbe := 0;
   Cold_Water_Temperature_Input.EnableAlarmMin := True;
   Cold_Water_Temperature_Input.EnableWarningMin := True;
   Cold_Water_Temperature_Input.EnableWarningMax := True;
   Cold_Water_Temperature_Input.EnableAlarmMax := True;
   Cold_Water_Temperature_Output.TypeProbe := 0;
   Cold_Water_Temperature_Output.EnableAlarmMin := True;
   Cold_Water_Temperature_Output.EnableWarningMin := True;
   Cold_Water_Temperature_Output.EnableWarningMax := True;
   Cold_Water_Temperature_Output.EnableAlarmMax := True;
   X_Axis_Temperature_PT1000.TypeProbe := 1;
   X_Axis_Temperature_PT1000.EnableAlarmMin := True;
   X_Axis_Temperature_PT1000.EnableWarningMin := True;
   X_Axis_Temperature_PT1000.EnableWarningMax := True;
   X_Axis_Temperature_PT1000.EnableAlarmMax := True;
   Y_Axis_Temperature_PT1000.TypeProbe := 1;
   Y_Axis_Temperature_PT1000.EnableAlarmMin := True;
   Y_Axis_Temperature_PT1000.EnableWarningMin := True;
   Y_Axis_Temperature_PT1000.EnableWarningMax := True;
   Y_Axis_Temperature_PT1000.EnableAlarmMax := True;
   X_Axis_Temperature_PTC.TypeProbe := 6;
   Y_Axis_Temperature_PTC.TypeProbe := 6;
   Nozzle_Overpressure.LimitUp := 10.0;
   Nozzle_Overpressure.LimitDown := 0.0;
   Nozzle_Overpressure.TypeProbe := 2;
   Nozzle_Overpressure.EnableAlarmMin := True;
   Nozzle_Overpressure.EnableWarningMin := True;
   Nozzle_Overpressure.EnableWarningMax := True;
   Nozzle_Overpressure.EnableAlarmMax := True;
   Optical_Path_Overpressure.LimitUp := 10.0;
   Optical_Path_Overpressure.LimitDown := 0.0;
   Optical_Path_Overpressure.TypeProbe := 2;
   Optical_Path_Overpressure.EnableAlarmMin := True;
   Optical_Path_Overpressure.EnableWarningMin := True;
   Optical_Path_Overpressure.EnableWarningMax := True;
   Optical_Path_Overpressure.EnableAlarmMax := True;
   Laser_Head_Overpressure.LimitUp := 10.0;
   Laser_Head_Overpressure.LimitDown := 0.0;
   Laser_Head_Overpressure.TypeProbe := 2;
   Laser_Head_Overpressure.EnableAlarmMin := True;
   Laser_Head_Overpressure.EnableWarningMin := True;
   Laser_Head_Overpressure.EnableWarningMax := True;
   Laser_Head_Overpressure.EnableAlarmMax := True;
   ZL_Axis_Overpressure.LimitUp := 10.0;
   ZL_Axis_Overpressure.LimitDown := 0.0;
   ZL_Axis_Overpressure.TypeProbe := 2;
   ZL_Axis_Overpressure.EnableAlarmMin := True;
   ZL_Axis_Overpressure.EnableWarningMin := True;
   ZL_Axis_Overpressure.EnableWarningMax := True;
   ZL_Axis_Overpressure.EnableAlarmMax := True;
   XY_Axis_Overpressure.LimitUp := 10.0;
   XY_Axis_Overpressure.LimitDown := 0.0;
   XY_Axis_Overpressure.TypeProbe := 2;
   XY_Axis_Overpressure.EnableAlarmMin := True;
   XY_Axis_Overpressure.EnableWarningMin := True;
   XY_Axis_Overpressure.EnableWarningMax := True;
   XY_Axis_Overpressure.EnableAlarmMax := True;
   Left_Aspiration.LimitUp := 2000.0;
   Left_Aspiration.LimitDown := 0.0;
   Left_Aspiration.TypeProbe := 5;
   Left_Aspiration.EnableAlarmMin := True;
   Left_Aspiration.EnableWarningMin := True;
   Left_Aspiration.EnableWarningMax := True;
   Left_Aspiration.EnableAlarmMax := True;
   Right_Aspiration.LimitUp := 2000.0;
   Right_Aspiration.LimitDown := 0.0;
   Right_Aspiration.TypeProbe := 5;
   Right_Aspiration.EnableAlarmMin := True;
   Right_Aspiration.EnableWarningMin := True;
   Right_Aspiration.EnableWarningMax := True;
   Right_Aspiration.EnableAlarmMax := True;
   Clim_Temperature.TypeProbe := 0;
   Sensor_Controller_Station1.LimitUp := 10.0;
   Sensor_Controller_Station1.LimitDown := -10.0;
   Sensor_Controller_Station1.TypeProbe := 3;
   Cabinet_Temperature.LimitUp := 50.0;
   Cabinet_Temperature.LimitDown := 0.0;
   Cabinet_Temperature.TypeProbe := 2;
END_DATA_BLOCK

DATA_BLOCK "DB_BadPartOnFixture"   // DB1308
{ S7_Optimized_Access := 'TRUE' }
// stored: AutoNumber false, MemoryReserve 100
   VAR
      BadPartOnFixture : Bool;
      ID_MeasureBad : Int;
   END_VAR
BEGIN
END_DATA_BLOCK

ORGANIZATION_BLOCK "Main"   // OB1, SCL, ProgramCycle
TITLE = "Main Program Sweep (Cycle)"
{ S7_Optimized_Access := 'TRUE' }
// stored: SetENOAutomatically false
   VAR_INPUT
      Initial_Call : Bool;   // Initial call of this OB
      Remanence : Bool;   // =True, if remanent data are available
   END_VAR
BEGIN
   REGION Description head
       //==================================================================================
       // POSALUX Swiss SA / (C) Copyright 2025
       //----------------------------------------------------------------------------------
       // Title: Main
       // Comment/Function: Cyclical execution of the program by the PLC
       // Author: Fabien WALDT
       // Engineering: TIA Portal v19
       //----------------------------------------------------------------------------------
       // Change log table:
       // Version  | Date     | Expert in charge | Changes applied
       //----------------------------------------------------------------------------------
       // 00.00.01 | 20250423 | WFA              | First released version
       //==================================================================================
   END_REGION

   REGION CNC
       // Call block for cyclical data exchange NC <-> PLC for the MCP
       "LBP_OpUnitComm_DB"(Config := "LBP_ConfigData");
       "LBP_MainBP"();
   END_REGION

   REGION IO
       "FC_AnalogInputsInit"();
       "DB_AnalogInputs"();
       "FC_AnalogInputAction"(iReset := "DB_McpKeyboardSignals".sAlarmReset.sKeySWStatus OR "MCP1_In".reset,
                              oBadPartOnFixture => "DB_BadPartOnFixture".BadPartOnFixture,
                              oID_MeasureBad=>"DB_BadPartOnFixture".ID_MeasureBad);
       "FC_AnalogInputConfig"();
       "DB_DigitalInputs"();
       "DB_DigitalInputsSonplas"();
       "DB_DigitalInputsBW_Station"();

       "DB_AnalogOutputs"();
       "DB_DigitalOutputs"();
       "DB_DigitalOutputsSonplas"();  
   END_REGION

   REGION Basic fonctions
       "DB_Impulsion"();
       "DB_ReadDateAndTime"();
   END_REGION

   REGION Interface PLC_ISO
       "DB_CommPLC_ISO"();
       "DB_MiscPLC_IHM_ISO"();
   END_REGION

   REGION SAFETY
       "FC_DataToSafety"();
       "DB_Alarms_Safety"();
   END_REGION

   REGION Load Unload Parts
       "DB_LoaderMain"();
       "DB_LoaderFixtureMain"();
       "DB_ExtraMissingPart"();
       "DB_PrioSequence"();
   END_REGION

   REGION Alarms
       "DB_Alarms"();

       "LBP_GenerateAlarmMsgs"(ToUserIF := true,
                               Quit := true,
                               NumActAlarmMsgs => "LBP_ConfigData".GenerateAlarmMsgs.NumActAlarmMsgs,
                               Error => "LBP_ConfigData".GenerateAlarmMsgs.Error,
                               StatusID => "LBP_ConfigData".GenerateAlarmMsgs.StatusID,
                               Status => "LBP_ConfigData".GenerateAlarmMsgs.Status);
       "DB_Msg"();
   END_REGION

   REGION Base Machine
       REGION Channel
           "DB_DecodChannels"();
           "DB_CycleStartStop"();
        END_REGION   

        REGION Axis
            "DB_Axis"();
            "DB_AxisPosition"();
        END_REGION

        REGION MCP
            "DB_MCPManagement"(); // Must be called after FC10 (LBP_GenerateAlarmMsgs)
        END_REGION

        REGION Laser
            "DB_LaserAirProcess"();
            "DB_LaserOperation"();
            "DB_LaserMeasureZoneSwitch"();  // WFA A Confirmer si plus utilisé
            "DB_Powermeter"();
        END_REGION

        REGION Air system
            "DB_Pressures"();
            "DB_Vacuums"();
        END_REGION

       REGION Vision
           "DB_Cognex"();
       END_REGION

       REGION Power Management
           "DB_Machineshutdown_UPS"();
           "DB_PowerOn"();
       END_REGION

       REGION Maintenance
           "DB_Maintenances"();
       END_REGION

       REGION Temperature Management
           "DB_Temperature"();
           "FC_ChillerMain"();
       END_REGION

       REGION Warm Up
           "DB_WarmUP"();
       END_REGION

       REGION Feed Override Display
           "DB_FeedOverride"(iA_FD_OR:="LBP_Chan1".A_FD_OR,
                             oFeedOverride=>"DB_FeedOverride".oFeedOverride);

       END_REGION
   END_REGION

   REGION Lights Management
       "DB_LightsManagement"();
   END_REGION

   REGION Main Door Management
       "DB_MainDoorManagement"();
   END_REGION

   REGION Config Machine
       "FC_GestionConfigMachine"();
   END_REGION

   REGION Tracability
       "DB_Tracability"(iCondTransfertExtInTo1:="DB_PartManagement".sPosition.sShuttle1.Undrilled.Presence.Part,
                        iCondTransfertExtInTo2:="DB_PartManagement".sPosition.sShuttle2.Undrilled.Presence.Part,
                        iCondTransfert1To3:="DB_LoaderShuttle1".sIntLoadUnload.oLoadGripperCloseReq,
                        iCondTransfert2To3:="DB_LoaderShuttle2".sIntLoadUnload.oLoadGripperCloseReq,
                        iCondTransfert3To4:="DB_PartManagement".sPosition.sFixture.Undrilled.Presence.Part,
                        iCondTransfert4To5:="DB_PartManagement".sPosition.sGripper.Drilled.Presence.Part,
                        iCondTransfert5To6:="DB_LoaderShuttle1".sIntLoadUnload.oUnloadGripperOpenReq,
                        iCondTransfert5To7:="DB_LoaderShuttle2".sIntLoadUnload.oUnloadGripperOpenReq,
                        iCondTransfert6ToExtOut:="DB_LoaderShuttle1".sExtLoadUnload.sInterface.JobDone AND NOT "DB_WorkingModes".sFilling,
                        iCondTransfert7ToExtOut:="DB_LoaderShuttle2".sExtLoadUnload.sInterface.JobDone AND NOT "DB_WorkingModes".sFilling);
   END_REGION

   REGION External Loader
       "DB_SonplasMain"();
   END_REGION

   REGION OPC
       // Keys
       "DB_HmiKeyboardSignals"();

       // Machine
       "DB_Parameters"();

       // Axis
       "DB_OPC_AxisManagement"();

       // State
       "DB_OPC_State"();

       // RealTime
       "DB_RealTime"();

       // Components
       "DB_Components"();

       // Laser
       "DB_Scanner"();
       "DB_Part_Data"();

       // Recipe
       "DB_Recipe"();
   END_REGION

   REGION Part Management
       "DB_PartManagement"();
   END_REGION

   REGION Bw loader
       "DB_BwLoader"();

   END_REGION

   REGION Working Modes
       "DB_GestionWorkingModes"();
   END_REGION

   REGION WAF A SUPPRIMER
       "DB_Simulation"();
   "DB_HMI_PLC_Pos"("HMI_Change Enable":=FALSE,
                    ioPLC_State:="DB_WAF".PLC_Pos,
                    ioHMI_State:="DB_WAF".HMI_Pos);
   END_REGION
END_ORGANIZATION_BLOCK

FUNCTION_BLOCK "FB_AnalogInputs"   // FB220, SCL
{ S7_Optimized_Access := 'FALSE' }
// stored: AutoNumber false, SetENOAutomatically false
   VAR
      sLaserPowerMeter : "FB_AnalogInput";
      sAxisB_ClampingPart : "FB_AnalogInput";
      sLaserAirPressureProcess : "FB_AnalogInput";
      sInletAirPressure : "FB_AnalogInput";
      sAmbiantTemperature : "FB_AnalogInput";
      sMachineTemperature : "FB_AnalogInput";
      sCold_WaterTemperatureInput : "FB_AnalogInput";
      sCold_WaterTemperatureOutput : "FB_AnalogInput";
      sX_AxisTemperaturePT1000 : "FB_AnalogInput";
      sY_AxisTemperaturePT1000 : "FB_AnalogInput";
      sX_AxisTemperaturePTC : "FB_AnalogInput";
      sY_AxisTemperaturePTC : "FB_AnalogInput";
      sNozzleOverpressure : "FB_AnalogInput";
      sOpticalPathOverpressure : "FB_AnalogInput";
      sLaserHeadOverpressure : "FB_AnalogInput";
      sZLAxisOverpressure : "FB_AnalogInput";
      sXYAxisOverpressure : "FB_AnalogInput";
      sLeftAspiration : "FB_AnalogInput";
      sRightAspiration : "FB_AnalogInput";
      sFreeIW458 : "FB_AnalogInput";
      sClimTemperature : "FB_AnalogInput";
      sFreeIW482 : "FB_AnalogInput";
      sFreeIW484 : "FB_AnalogInput";
      sFreeIW486 : "FB_AnalogInput";
      sSensorControllerStation1 : "FB_AnalogInput";
      sCabinetTemperature : "FB_AnalogInput";
      sFreeIW464 : "FB_AnalogInput";
      sFreeIW466 : "FB_AnalogInput";
   END_VAR
   VAR_TEMP
      tAlarm_OutOfRange : Bool;
      tDummyLimit : Real;
   END_VAR
BEGIN
   REGION Description header 
       //==================================================================================
       // POSALUX Swiss SA / (C) Copyright 2025
       //----------------------------------------------------------------------------------
       // Title: Analog Inputs Configuration 
       // Comment/Function: Configuration of analog inputs
       // Author: Fabien WALDT
       // Engineering: TIA Portal v17
       //----------------------------------------------------------------------------------
       // Change log table:
       // Version  | Date     | Expert in charge | Changes applied
       // ---------|----------|------------------|-----------------------------------------
       // 00.00.01 | 20250423 | WFA              | First released version
       // =================================================================================
   END_REGION

   // ET200SP Mapping
   REGION IW412 - IW418 : AI 4xU/I 2-wire ST Slot 9
       #sLaserPowerMeter(iValueHW := "AI_LaserPowerMeter",
                         iID := 701,
                         iHMI_UpdateEnable := TRUE,
                         ioDataHMI := "DB_AnalogInputDataHMI".Laser_Power_Meter,
                         ioAlarmOutOfRange := #tAlarm_OutOfRange,
                         ioDataPLC := "DB_AnalogInputDataPLC".Laser_Power_Meter,
                         ioOPC := "DB_OPC_AnalogInputs".Signals[1]);

       #sAxisB_ClampingPart(iValueHW :="AI_AxisB_ClampingPart",
                            iID:= 810,
                            iHMI_UpdateEnable:= TRUE,
                            ioDataHMI:= "DB_AnalogInputDataHMI".Axis_B_Clamping_Part,
                            ioAlarmOutOfRange := #tAlarm_OutOfRange,
                            ioDataPLC := "DB_AnalogInputDataPLC".Axis_B_Clamping_Part,
                            ioOPC:= "DB_OPC_AnalogInputs".Signals[2]);

       #sLaserAirPressureProcess(iValueHW :="AI_LaserAirPressureProcess",
                                 iID:= 511,
                                 iHMI_UpdateEnable:= TRUE,
                                 ioDataHMI:= "DB_AnalogInputDataHMI".Laser_Air_Pressure_Process,
                                 ioAlarmOutOfRange := #tAlarm_OutOfRange,
                                 ioDataPLC := "DB_AnalogInputDataPLC".Laser_Air_Pressure_Process,
                                 ioOPC:= "DB_OPC_AnalogInputs".Signals[3]);

       #sInletAirPressure(iValueHW :="AI_InletAirPressure",
                          iID:= 501,
                          iHMI_UpdateEnable:= TRUE,
                          ioDataHMI:= "DB_AnalogInputDataHMI".Inlet_Air_Pressure,
                          ioAlarmOutOfRange := "LBP_AlarmMsgs".UserA[01].A70UUxx[03],
                          ioDataPLC := "DB_AnalogInputDataPLC".Inlet_Air_Pressure,
                          ioOPC:= "DB_OPC_AnalogInputs".Signals[4]);
   END_REGION

   REGION IW420 - IW426 : AI4 x RTD/TC HF Slot 10
       #sAmbiantTemperature(iValueHW := "AI_AmbiantTemperature",
                            iID:= 201,
                            iHMI_UpdateEnable:= TRUE,
                            ioDataHMI:= "DB_AnalogInputDataHMI".Ambiant_Temperature,
                            ioAlarmOutOfRange := "LBP_AlarmMsgs".UserA[01].A70UUxx[08],
                            ioDataPLC := "DB_AnalogInputDataPLC".Ambiant_Temperature,
                            ioOPC:= "DB_OPC_AnalogInputs".Signals[5]);

       #sMachineTemperature(iValueHW := "AI_MachineTemperature",
                            iID:= 202,
                            iHMI_UpdateEnable:= TRUE,
                            ioDataHMI:= "DB_AnalogInputDataHMI".Machine_Temperature,
                            ioAlarmOutOfRange := "LBP_AlarmMsgs".UserA[01].A70UUxx[09],
                            ioDataPLC := "DB_AnalogInputDataPLC".Machine_Temperature,
                            ioOPC:= "DB_OPC_AnalogInputs".Signals[6]);

       #sCold_WaterTemperatureInput(iValueHW := "AI_ColdWaterTemperatureInput",
                                    iID:= 301,
                                    iHMI_UpdateEnable:= TRUE,
                                    ioDataHMI:= "DB_AnalogInputDataHMI".Cold_Water_Temperature_Input,
                                    ioAlarmOutOfRange := "LBP_AlarmMsgs".UserA[01].A70UUxx[10],
                                    ioDataPLC := "DB_AnalogInputDataPLC".Cold_Water_Temperature_Input,
                                    ioOPC:= "DB_OPC_AnalogInputs".Signals[7]);

       #sCold_WaterTemperatureOutput(iValueHW := "AI_ColdWaterTemperatureOutput",
                                     iID:= 302,
                                     iHMI_UpdateEnable:= TRUE,
                                     ioDataHMI:= "DB_AnalogInputDataHMI".Cold_Water_Temperature_Output,
                                     ioAlarmOutOfRange := "LBP_AlarmMsgs".UserA[01].A70UUxx[11],
                                     ioDataPLC := "DB_AnalogInputDataPLC".Cold_Water_Temperature_Output,
                                     ioOPC:= "DB_OPC_AnalogInputs".Signals[8]);
   END_REGION

   REGION IW436 - IW442 : AI4 x RTD/TC HF Slot 11
       #sX_AxisTemperaturePT1000(iValueHW := "AI_X_AxisTemperaturePT1000",
                                 iID:= 110,
                                 iHMI_UpdateEnable:= TRUE,
                                 ioDataHMI:= "DB_AnalogInputDataHMI".X_Axis_Temperature_PT1000,
                                 ioAlarmOutOfRange := "LBP_AlarmMsgs".UserA[01].A70UUxx[12],
                                 ioDataPLC := "DB_AnalogInputDataPLC".X_Axis_Temperature_PT1000,
                                 ioOPC:= "DB_OPC_AnalogInputs".Signals[9]);

       #sY_AxisTemperaturePT1000(iValueHW := "AI_Y_AxisTemperaturePT1000",
                                 iID:= 120,
                                 iHMI_UpdateEnable:= TRUE,
                                 ioDataHMI:= "DB_AnalogInputDataHMI".Y_Axis_Temperature_PT1000,
                                 ioAlarmOutOfRange := "LBP_AlarmMsgs".UserA[01].A70UUxx[13],
                                 ioDataPLC := "DB_AnalogInputDataPLC".Y_Axis_Temperature_PT1000,
                                 ioOPC:= "DB_OPC_AnalogInputs".Signals[10]);

       #sX_AxisTemperaturePTC(iValueHW := "AI_X_ AxisTemperaturePTC",
                              iID:= 116,
                              iHMI_UpdateEnable:= TRUE,
                              ioDataHMI:= "DB_AnalogInputDataHMI".X_Axis_Temperature_PTC,
                              ioAlarmOutOfRange := "LBP_AlarmMsgs".UserA[01].A70UUxx[14],
                              ioDataPLC := "DB_AnalogInputDataPLC".X_Axis_Temperature_PTC,
                              ioOPC:= "DB_OPC_AnalogInputs".Signals[11]);

       #sY_AxisTemperaturePTC(iValueHW := "AI_Y_ AxisTemperaturePTC",
                              iID:= 126,
                              iHMI_UpdateEnable:= TRUE,
                              ioDataHMI:= "DB_AnalogInputDataHMI".Y_Axis_Temperature_PTC,
                              ioAlarmOutOfRange := "LBP_AlarmMsgs".UserA[01].A70UUxx[15],
                              ioDataPLC := "DB_AnalogInputDataPLC".Y_Axis_Temperature_PTC,
                              ioOPC:= "DB_OPC_AnalogInputs".Signals[12]);
   END_REGION

   REGION IW444 - IW458 : AI8 x U BA Slot 12
       #sNozzleOverpressure(iValueHW := "AI_NozzleOverpressure",
                            iID:= 512,
                            iHMI_UpdateEnable:= TRUE,
                            ioDataHMI:= "DB_AnalogInputDataHMI".Nozzle_Overpressure,
                            ioAlarmOutOfRange := #tAlarm_OutOfRange,
                            ioDataPLC := "DB_AnalogInputDataPLC".Nozzle_Overpressure,
                            ioOPC:= "DB_OPC_AnalogInputs".Signals[13]);

       #sOpticalPathOverpressure(iValueHW := "AI_OpticalPathOverpressure",
                                 iID:= 513,
                                 iHMI_UpdateEnable:= TRUE,
                                 ioDataHMI:= "DB_AnalogInputDataHMI".Optical_Path_Overpressure,
                                 ioAlarmOutOfRange := "LBP_AlarmMsgs".UserA[01].A70UUxx[05],
                                 ioDataPLC := "DB_AnalogInputDataPLC".Optical_Path_Overpressure,
                                 ioOPC:= "DB_OPC_AnalogInputs".Signals[14]);

       #sLaserHeadOverpressure(iValueHW := "AI_LaserHeadOverpressure",
                               iID:= 514,
                               iHMI_UpdateEnable:= TRUE,
                               ioDataHMI:= "DB_AnalogInputDataHMI".Laser_Head_Overpressure,
                               ioAlarmOutOfRange := "LBP_AlarmMsgs".UserA[01].A70UUxx[06],
                               ioDataPLC := "DB_AnalogInputDataPLC".Laser_Head_Overpressure,
                               ioOPC:= "DB_OPC_AnalogInputs".Signals[15]);

       #sZLAxisOverpressure(iValueHW := "AI_ZL_AxisOverpressure",
                            iID:= 520,
                            iHMI_UpdateEnable:= TRUE,
                            ioDataHMI:= "DB_AnalogInputDataHMI".ZL_Axis_Overpressure,
                            ioAlarmOutOfRange := "LBP_AlarmMsgs".UserA[01].A70UUxx[04],
                            ioDataPLC := "DB_AnalogInputDataPLC".ZL_Axis_Overpressure,
                            ioOPC:= "DB_OPC_AnalogInputs".Signals[16]);

       #sXYAxisOverpressure(iValueHW := "AI_XY_AxisOverpressure",
                            iID:= 530,
                            iHMI_UpdateEnable:= TRUE,
                            ioDataHMI:= "DB_AnalogInputDataHMI".XY_Axis_Overpressure,
                            ioAlarmOutOfRange := "LBP_AlarmMsgs".UserA[01].A70UUxx[07],
                            ioDataPLC := "DB_AnalogInputDataPLC".XY_Axis_Overpressure,
                            ioOPC:= "DB_OPC_AnalogInputs".Signals[17]);

       #sLeftAspiration(iValueHW := "AI_LeftAspiration",
                        iID:= 401,
                        iHMI_UpdateEnable:= TRUE,
                        ioDataHMI:= "DB_AnalogInputDataHMI".Left_Aspiration,
                        ioAlarmOutOfRange := #tAlarm_OutOfRange,
                        ioDataPLC := "DB_AnalogInputDataPLC".Left_Aspiration,
                        ioOPC:= "DB_OPC_AnalogInputs".Signals[18]);

       #sRightAspiration(iValueHW := "AI_RightAspiration",
                         iID:= 402,
                         iHMI_UpdateEnable:= TRUE,
                         ioDataHMI:= "DB_AnalogInputDataHMI".Right_Aspiration,
                         ioAlarmOutOfRange := #tAlarm_OutOfRange,
                         ioDataPLC := "DB_AnalogInputDataPLC".Right_Aspiration,
                         ioOPC:= "DB_OPC_AnalogInputs".Signals[19]);

       #sFreeIW458(iValueHW := "AI_FreeIW458",
                   iID:= 999,
                   iHMI_UpdateEnable:= TRUE,
                   ioDataHMI:= "DB_AnalogInputDataHMI".Free_IW458,
                   ioAlarmOutOfRange := #tAlarm_OutOfRange,
                   ioDataPLC := "DB_AnalogInputDataPLC".Free_IW458,
                   ioOPC:= "DB_OPC_AnalogInputs".Signals[20]);
   END_REGION

   REGION IW480 - IW486 : AI4 x RTD/TC HF Slot 12
       #sClimTemperature(iValueHW := "AI_ClimTemperature",
                         iID:= 204,
                         iHMI_UpdateEnable:= TRUE,
                         ioDataHMI:= "DB_AnalogInputDataHMI".Clim_Temperature,
                         ioAlarmOutOfRange := #tAlarm_OutOfRange,
                         ioDataPLC := "DB_AnalogInputDataPLC".Clim_Temperature,
                         ioOPC:="DB_OPC_AnalogInputs".Signals[21]);

       #sFreeIW482(iValueHW := "AI_FreeIW482",
                   iID:= 999,
                   iHMI_UpdateEnable:=TRUE,
                   ioDataHMI:= "DB_AnalogInputDataHMI".Free_IW482,
                   ioAlarmOutOfRange := #tAlarm_OutOfRange,
                   ioDataPLC := "DB_AnalogInputDataPLC".Free_IW482,
                   ioOPC:= "DB_OPC_AnalogInputs".Signals[22]);

       #sFreeIW484(iValueHW := "AI_FreeIW484",
                   iID:= 999,
                   iHMI_UpdateEnable:= TRUE,
                   ioDataHMI:= "DB_AnalogInputDataHMI".Free_IW484,
                   ioAlarmOutOfRange := #tAlarm_OutOfRange,
                   ioDataPLC := "DB_AnalogInputDataPLC".Free_IW484,
                   ioOPC:= "DB_OPC_AnalogInputs".Signals[23]);

       #sFreeIW486(iValueHW := "AI_FreeIW486",
                   iID:= 999,
                   iHMI_UpdateEnable:= TRUE,
                   ioDataHMI:= "DB_AnalogInputDataHMI".Free_IW486,
                   ioAlarmOutOfRange := #tAlarm_OutOfRange,
                   ioDataPLC := "DB_AnalogInputDataPLC".Free_IW486,
                   ioOPC:= "DB_OPC_AnalogInputs".Signals[24]);
   END_REGION

   REGION IW500 - IW514 : AI 4xU/I 2-wire ST Slot 21
       #sSensorControllerStation1(iValueHW := "AI_SensorControllerStation1",
                                  iID:= 711,
                                  iHMI_UpdateEnable:= TRUE,
                                  ioDataHMI:= "DB_AnalogInputDataHMI".Sensor_Controller_Station1,
                                  ioAlarmOutOfRange := #tAlarm_OutOfRange,
                                  ioDataPLC := "DB_AnalogInputDataPLC".Sensor_Controller_Station1,
                                  ioOPC:= "DB_OPC_AnalogInputs".Signals[25]);

       #sCabinetTemperature(iValueHW := "AI_CabinetTemperature",
                            iID:= 203,
                            iHMI_UpdateEnable:= TRUE,
                            ioDataHMI:= "DB_AnalogInputDataHMI".Cabinet_Temperature,
                            ioAlarmOutOfRange := "LBP_AlarmMsgs".UserA[01].A70UUxx[20],
                            ioDataPLC := "DB_AnalogInputDataPLC".Cabinet_Temperature,
                            ioOPC:= "DB_OPC_AnalogInputs".Signals[26]);

       #sFreeIW464(iValueHW := "AI_FreeIW464",
                   iID:= 999,
                   iHMI_UpdateEnable:= TRUE,
                   ioDataHMI:= "DB_AnalogInputDataHMI".Free_IW464,
                   ioAlarmOutOfRange := #tAlarm_OutOfRange,
                   ioDataPLC := "DB_AnalogInputDataPLC".Free_IW464,
                   ioOPC:= "DB_OPC_AnalogInputs".Signals[27]);

       #sFreeIW466(iValueHW := "AI_FreeIW466",
                   iID:= 999,
                   iHMI_UpdateEnable:= TRUE,
                   ioDataHMI:= "DB_AnalogInputDataHMI".Free_IW466,
                   ioAlarmOutOfRange := #tAlarm_OutOfRange,
                   ioDataPLC := "DB_AnalogInputDataPLC".Free_IW466,
                   ioOPC:= "DB_OPC_AnalogInputs".Signals[28]);
   END_REGION
END_FUNCTION_BLOCK

FUNCTION_BLOCK "FB_AnalogInput"   // FB10, SCL
{ S7_Optimized_Access := 'FALSE' }
// stored: AutoNumber false, SetENOAutomatically false
   VAR_INPUT
      iValueHW { ExternalAccessible := 'False'; ExternalVisible := 'False'; ExternalWritable := 'False'} : Word;   // Value in word from PLC analog input
      iID : Int;
      iHMI_UpdateEnable : Bool;
   END_VAR
   VAR_IN_OUT
      ioAlarmOutOfRange { ExternalAccessible := 'False'; ExternalVisible := 'False'; ExternalWritable := 'False'} : Bool;   // Hardware signal out of nominal range alarm
      ioDataPLC : "AnalogInDataPLC_DT";
      ioDataHMI : "AnalogInDataHMI_DT";
      ioOPC : "UDT_OPC_Analog";
   END_VAR
   VAR
      sSWRealValue { ExternalAccessible := 'False'; ExternalVisible := 'False'; ExternalWritable := 'False'} : Real;
      sRT_Clock_1Hz : R_TRIG;
      sDownload { S7_SetPoint := 'True'} : Bool;   // Download DataHMI to OPC
   END_VAR
   VAR_TEMP
      tActual_input_value : Real;
   END_VAR
   VAR CONSTANT
      PT100 : UInt := 0;
      PT1000 : UInt := 1;
      TYP_0_10V : UInt := 2;
      "TYP_-10_10V" : UInt := 3;
      RES600 : UInt := 4;
      SL5201 : UInt := 5;
      PTC : UInt := 6;
   END_VAR
BEGIN
   REGION Description header 
       //==================================================================================
       // POSALUX Swiss SA / (C) Copyright 2025
       //----------------------------------------------------------------------------------
       // Title: AI_Alloc
       // Comment/Function:  Analog input management :  
       //                       - Based on input type (PT100, PT1000, 0-10V, -10+10V, RES600)  
       //                       - Value correction capability (y = Ax + B)  
       //                       - Alarm generation if measurement is out of tolerance (Alarm reset in FB_alarms)
       //                       - OPC Communication
       // Author: Fabien Waldt
       // Engineering: TIA Portal v17
       //----------------------------------------------------------------------------------
       // Change log table:
       // Version  | Date     | Expert in charge | Changes applied
       // ---------|----------|------------------|------------------------------------
       // 00.00.01 | 20250304 | FWA              | First released version
       // 00.00.02 | 20250610 | GSR              | Correction iAxFactor/iBOffset
       // 00.00.03 | 20251114 | FWA              | Add OPC Features
       // ==================================================================================
   END_REGION


   REGION Type of Probe
       CASE #ioDataPLC.TypeProbe OF
           #PT100:
               IF WORD_TO_INT(#iValueHW) <= 800 AND WORD_TO_INT(#iValueHW) >= -2000 THEN
                   #tActual_input_value := (INT_TO_REAL(WORD_TO_INT(#iValueHW)) * 0.1)*#ioDataHMI.AxFactor;
               ELSE
                   #tActual_input_value := 0.0;
                   #ioAlarmOutOfRange := TRUE;
               END_IF;

           #PT1000:
               IF WORD_TO_INT(#iValueHW) <= 800 AND WORD_TO_INT(#iValueHW) >= -2000 THEN
                   #tActual_input_value := (INT_TO_REAL(WORD_TO_INT(#iValueHW)) * 0.1)*#ioDataHMI.AxFactor;
               ELSE
                   #tActual_input_value := 0.0;
                   #ioAlarmOutOfRange := TRUE;
               END_IF;

           #TYP_0_10V:
               IF #iValueHW <= 27648 AND #iValueHW >= 0 THEN
                   #tActual_input_value := (((INT_TO_REAL(WORD_TO_INT(#iValueHW))*#ioDataHMI.AxFactor) * (#ioDataPLC.LimitUp - #ioDataPLC.LimitDown)) / 27648.0) *#ioDataHMI.AxFactor;
               ELSE
                   #tActual_input_value := 0.0;
                   #ioAlarmOutOfRange := TRUE;
               END_IF;

           #"TYP_-10_10V":
               IF (WORD_TO_INT(#iValueHW) <= 32767) AND (WORD_TO_INT(#iValueHW) >= -32767) THEN
                   #tActual_input_value := (((INT_TO_REAL(WORD_TO_INT(#iValueHW)) + 32767) * (#ioDataPLC.LimitUp - #ioDataPLC.LimitDown) / (2 * 32767))) *#ioDataHMI.AxFactor + #ioDataPLC.LimitDown;
               ELSE
                   #tActual_input_value := 0.0;
                   #ioAlarmOutOfRange := TRUE;
               END_IF;

           #RES600:
               IF #iValueHW <= 27648 AND #iValueHW >= 0 THEN
                   #tActual_input_value := (((INT_TO_REAL(WORD_TO_INT(#iValueHW))*#ioDataHMI.AxFactor) * (#ioDataPLC.LimitUp - #ioDataPLC.LimitDown)) / 27648.0) *#ioDataHMI.AxFactor ;
               ELSE
                   #tActual_input_value := 0.0;
                   #ioAlarmOutOfRange := TRUE;
               END_IF;
           #SL5201:
               IF #iValueHW <= 27648 AND #iValueHW >= 0 THEN
                   #tActual_input_value := (LREAL_TO_REAL(1.4774 * EXP(0.2536 * (WORD_TO_INT(#iValueHW) * 10.0 / 27648.0))))*#ioDataHMI.AxFactor;
               ELSE
                   #tActual_input_value := 0.0;
                   #ioAlarmOutOfRange := TRUE;
               END_IF;
           #PTC:
               IF #iValueHW.%X7 AND NOT #iValueHW.%X0 AND NOT #iValueHW.%X2 THEN
                   // Reaction to short-circuit : < 18 Ω -> SIMATIC S7: Bit 7 (IB x+1) = "1", Bit 0 = "0" and Bit 2 = "0"
                   // See documentation: Analog input module AI 4xRTD/TC 2-/3-/4-wire HF (6ES7134-6JD00-0CA1)
                   #ioAlarmOutOfRange := TRUE;
               ELSE
                   // No measurement value for PTC analog input ' bits 0 and 2 are handled in the related FB (Temperature)
                   // Normal range: < 550 Ω             -> Bit 0 = "0", Bit 2 = "0"
                   // Prewarning range: 550 Ω to 1650 Ω -> Bit 0 = "0", Bit 2 = "1"
                   // Response range: > 1650 Ω          -> Bit 0 = "1", Bit 2 = "0"
                   // See documentation Analog input module AI 4xRTD/TC 2-/3-/4-wire HF (6ES7134-6JD00-0CA1)
                   #tActual_input_value := (WORD_TO_INT(#iValueHW))*#ioDataHMI.AxFactor;
               END_IF;
       END_CASE;
   END_REGION

   REGION Update Values
       #sSWRealValue := #tActual_input_value + #ioDataHMI.BOffset;
       #ioDataHMI.CurrentValue := #sSWRealValue;
   END_REGION

   REGION OPC
       IF #ioOPC.Update AND #iHMI_UpdateEnable THEN
           // Copy HMI parameters (from OPC Parameters IHM) to HMI Datas (Used in PLC program)
           #ioDataHMI.StartTime := DINT_TO_TIME(REAL_TO_DINT(#ioOPC.Delay))*1000;
           #ioDataHMI.ThresholdAlarmMax := #ioOPC.DiffErrorMax;
           #ioDataHMI.ThresholdAlarmMin := #ioOPC.DiffErrorMin;
           #ioDataHMI.ThresholdWarningMax := #ioOPC.DiffWarnMax;
           #ioDataHMI.ThresholdWarningMin := #ioOPC.DiffWarnMin;
           #ioDataHMI.BOffset := #ioOPC.Offset;
           // #ioDataHMI.AxFactor := #ioOPC.Parameters.Gain; // Currently not on HMI
           #ioDataHMI.TargetValue := #ioOPC.Target;

           // Copy HMI Datas (Used in PLC program) to HMI (OPC Display HMI)
           #ioOPC.Delay := DINT_TO_REAL(TIME_TO_DINT(#ioDataHMI.StartTime)) / 1000.0;
           #ioOPC.DiffErrorMax := #ioDataHMI.ThresholdAlarmMax;
           #ioOPC.DiffErrorMin := #ioDataHMI.ThresholdAlarmMin;
           #ioOPC.DiffWarnMax := #ioDataHMI.ThresholdWarningMax;
           #ioOPC.DiffWarnMin := #ioDataHMI.ThresholdWarningMin;
           #ioOPC.Offset := #ioDataHMI.BOffset;
           // #ioOPC.Gain := #ioDataHMI.AxFactor; // Currently not on HMI
           #ioOPC.Target := #ioDataHMI.TargetValue;
           #ioOPC.Update := FALSE;
       END_IF;

       // Update ID
       #ioDataHMI.ID_Measure := #iID;
       #ioOPC.Id := #ioDataHMI.ID_Measure;

       // Update Current Value
       #sRT_Clock_1Hz(CLK := "Clock_1Hz");
       IF #sRT_Clock_1Hz.Q THEN
           #ioOPC.Value := #ioDataHMI.CurrentValue;
       END_IF;

       // Download DataHMI to OPC (Only used to initialize OPC Datas)
       IF #sDownload THEN
           // Copy HMI Datas (Used in PLC program) to HMI (OPC Display HMI)
           #ioOPC.Delay := DINT_TO_REAL(TIME_TO_DINT(#ioDataHMI.StartTime))/1000.0;
           #ioOPC.DiffErrorMax := #ioDataHMI.ThresholdAlarmMax;
           #ioOPC.DiffErrorMin := #ioDataHMI.ThresholdAlarmMin;
           #ioOPC.DiffWarnMax := #ioDataHMI.ThresholdWarningMax;
           #ioOPC.DiffWarnMin := #ioDataHMI.ThresholdWarningMin;
           #ioOPC.Offset := #ioDataHMI.BOffset;
           // #ioOPC.Gain := #ioDataHMI.AxFactor; // Currently not on HMI
           #ioOPC.Target := #ioDataHMI.TargetValue;
           #sDownload := FALSE;
       END_IF;
   END_REGION
END_FUNCTION_BLOCK

FUNCTION_BLOCK "FB_DigitalInputs"   // FB210, SCL
{ S7_Optimized_Access := 'TRUE' }
// stored: AutoNumber false, MemoryReserve 100, SetENOAutomatically false
   VAR
      sFreeI0_0 : "FB_DigitalInput";
      sX_AxisBrakePressCtrl : "FB_DigitalInput";
      sY_AxisBrakePressCtrl : "FB_DigitalInput";
      sBreakerCtrl : "FB_DigitalInput";
      sCabinetTemperatureCtrl : "FB_DigitalInput";
      sUPS_PowerFailure : "FB_DigitalInput";
      sAirPressureCtrl : "FB_DigitalInput";
      sShutterClosed : "FB_DigitalInput";
      sAirDryerOK : "FB_DigitalInput";
      sUPS_BatteryOK : "FB_DigitalInput";
      sFrontDoorClosed : "FB_DigitalInput";
      sInfeedReadyOK_Start : "FB_DigitalInput";
      sCoolingOK : "FB_DigitalInput";
      sFreeI1_5 : "FB_DigitalInput";
      sPowerReady : "FB_DigitalInput";
      sAlarmI2T : "FB_DigitalInput";
      sHeadLaserBusy : "FB_DigitalInput";
      sHeadLaserBreaker { S7_SetPoint := 'True'} : "FB_DigitalInput";
      sFrontDoorLocked { S7_SetPoint := 'True'} : "FB_DigitalInput";
      sUPS_CommonAlarm { S7_SetPoint := 'True'} : "FB_DigitalInput";
      sUPS_BatteryLow { S7_SetPoint := 'True'} : "FB_DigitalInput";
      sFreeI2_5 { S7_SetPoint := 'True'} : "FB_DigitalInput";
      sHeadChillerHighPressure { S7_SetPoint := 'True'} : "FB_DigitalInput";
      sHeadChillerWaterTemperature { S7_SetPoint := 'True'} : "FB_DigitalInput";
      sHeadChillerFlow { S7_SetPoint := 'True'} : "FB_DigitalInput";
      sHeadChillerCollectivFault { S7_SetPoint := 'True'} : "FB_DigitalInput";
      sHeadChillerWaterLevel { S7_SetPoint := 'True'} : "FB_DigitalInput";
      sUPS_ByPassActive { S7_SetPoint := 'True'} : "FB_DigitalInput";
      sHeadChillerAmbiantTemperature { S7_SetPoint := 'True'} : "FB_DigitalInput";
      sFreeI3_5 { S7_SetPoint := 'True'} : "FB_DigitalInput";
      sFreeI3_6 { S7_SetPoint := 'True'} : "FB_DigitalInput";
      sFreeI3_7 { S7_SetPoint := 'True'} : "FB_DigitalInput";
      sLoadClampOpened { S7_SetPoint := 'True'} : "FB_DigitalInput";
      sLoadClampNotClosedWithPart { S7_SetPoint := 'True'} : "FB_DigitalInput";
      sUnloadClampOpened { S7_SetPoint := 'True'} : "FB_DigitalInput";
      sUPS_Fault { S7_SetPoint := 'True'} : "FB_DigitalInput";
      sInternalGateLocked { S7_SetPoint := 'True'} : "FB_DigitalInput";
      sExternalGateLocked { S7_SetPoint := 'True'} : "FB_DigitalInput";
      sInverterActive { S7_SetPoint := 'True'} : "FB_DigitalInput";
      sUnloadClampNotClosedWithPart { S7_SetPoint := 'True'} : "FB_DigitalInput";
      sFreeI5_0 { S7_SetPoint := 'True'} : "FB_DigitalInput";
      sFreeI5_1 { S7_SetPoint := 'True'} : "FB_DigitalInput";
      sInternalGateOpened { S7_SetPoint := 'True'} : "FB_DigitalInput";
      sExternalGateOpened { S7_SetPoint := 'True'} : "FB_DigitalInput";
      sPowerMeterBackCtrl { S7_SetPoint := 'True'} : "FB_DigitalInput";
      sPowerMeterFrontCtrl { S7_SetPoint := 'True'} : "FB_DigitalInput";
      sFreeI5_6 { S7_SetPoint := 'True'} : "FB_DigitalInput";
      sFreeI5_7 { S7_SetPoint := 'True'} : "FB_DigitalInput";
      sHeadChillerCutOff { S7_SetPoint := 'True'} : "FB_DigitalInput";
      sHeadChillerTemperature { S7_SetPoint := 'True'} : "FB_DigitalInput";
      sFreeI6_2 { S7_SetPoint := 'True'} : "FB_DigitalInput";
      sFreeI6_3 { S7_SetPoint := 'True'} : "FB_DigitalInput";
      sClampingOpenCtrl { S7_SetPoint := 'True'} : "FB_DigitalInput";
      sB_Axis_BrakeReleasedCtrl { S7_SetPoint := 'True'} : "FB_DigitalInput";
      sFreeI6_6 { S7_SetPoint := 'True'} : "FB_DigitalInput";
      sB_AxisReferencePoint { S7_SetPoint := 'True'} : "FB_DigitalInput";
      sSourceChillerHighPressure { S7_SetPoint := 'True'} : "FB_DigitalInput";
      sSourceChillerWaterTemperature { S7_SetPoint := 'True'} : "FB_DigitalInput";
      sSourceChillerFlow { S7_SetPoint := 'True'} : "FB_DigitalInput";
      sSourceChillerCollectivFault { S7_SetPoint := 'True'} : "FB_DigitalInput";
      sSourceChillerWaterLevel { S7_SetPoint := 'True'} : "FB_DigitalInput";
      sSourceChillerAmbiantTemperature { S7_SetPoint := 'True'} : "FB_DigitalInput";
      sSourceChillerCutOff { S7_SetPoint := 'True'} : "FB_DigitalInput";
      sSourceChillerTemperature { S7_SetPoint := 'True'} : "FB_DigitalInput";
   END_VAR
BEGIN
   REGION Description head
       //==================================================================================
       // POSALUX Swiss SA / (C) Copyright 2025
       //----------------------------------------------------------------------------------
       // Title: Digital Inputs mapping
       // Comment/Function: Digital Inputs mapping
       // Author: Fabien WALDT
       // Engineering: TIA Portal v17
       //----------------------------------------------------------------------------------
       // Change log table:
       // Version  | Date     | Expert in charge | Changes applied
       // ---------|----------|------------------|-----------------------------------------
       // 00.00.01 | 20250423 | WFA              | First released version
       // =================================================================================
   END_REGION

       // ET200SP Mapping
   REGION I0.0 - I1.7 : DI 16x24VDC ST Slot 1
       #sFreeI0_0(iHWStatus := "DI_FreeI0_0");
       #sX_AxisBrakePressCtrl(iHWStatus := "DI_X_AxisBrakePressCtrl");
       #sY_AxisBrakePressCtrl(iHWStatus := "DI_Y_AxisBrakePressCtrl");
       #sBreakerCtrl(iHWStatus := "DI_BreakerCtrl");
       #sCabinetTemperatureCtrl(iHWStatus := "DI_CabinetTemperatureCtrl");
       #sUPS_PowerFailure(iHWStatus := "DI_UPS_PowerFailure");
       #sAirPressureCtrl(iHWStatus := "DI_AirPressureCtrl");
       #sShutterClosed(iHWStatus := "DI_ShutterClosed");
       //
       #sAirDryerOK(iHWStatus := "DI_AirDryerOK");
       #sUPS_BatteryOK(iHWStatus := "DI_UPS_BatteryOK");
       #sFrontDoorClosed(iHWStatus := "DI_FrontDoorClosed");
       #sInfeedReadyOK_Start(iHWStatus := "DI_InfeedReadyOK_Start");
       #sCoolingOK(iHWStatus := "DI_CoolingOK");
       #sFreeI1_5(iHWStatus := "DI_FreeI1_5");
       #sPowerReady(iHWStatus := "DI_PowerReady");
       #sAlarmI2T(iHWStatus := "DI_AlarmI2T");
   END_REGION

   REGION I2.0 - I3.7 : DI 16x24VDC ST Slot 2
       #sHeadLaserBusy(iHWStatus := "DI_HeadLaserBusy");
       #sHeadLaserBreaker(iHWStatus := "DI_HeadLaserBreaker");
       #sFrontDoorLocked(iHWStatus := "DI_FrontDoorLocked");
       #sUPS_CommonAlarm(iHWStatus := "DI_UPS_CommonAlarm");
       #sUPS_BatteryLow(iHWStatus := "DI_UPS_BatteryLow");
       #sFreeI2_5(iHWStatus := "DI_FreeI2_5");
       #sHeadChillerHighPressure(iHWStatus := "DI_HeadChillerHighPressure");
       #sHeadChillerWaterTemperature(iHWStatus := "DI_HeadChillerWaterTemperature");
       //
       #sHeadChillerFlow(iHWStatus := "DI_HeadChillerFlow");
       #sHeadChillerCollectivFault(iHWStatus := "DI_HeadChillerCollectivFault");
       #sHeadChillerWaterLevel(iHWStatus := "DI_HeadChillerWaterLevel");
       #sUPS_ByPassActive(iHWStatus := "DI_UPSByPassActive");
       #sHeadChillerAmbiantTemperature(iHWStatus := "DI_HeadChillerAmbiantTemperature");
       #sFreeI3_5(iHWStatus := "DI_FreeI3_5");
       #sFreeI3_6(iHWStatus := "DI_FreeI3_6");
       #sFreeI3_7(iHWStatus := "DI_FreeI3_7");
   END_REGION

   REGION I4.0 - I5.7 : DI 16x24VDC ST Slot 3
       #sLoadClampOpened(iHWStatus := "DI_LoadClampOpened");
       #sLoadClampNotClosedWithPart(iHWStatus := "DI_LoadClampNotClosedWithPart");
       #sUnloadClampOpened(iHWStatus := "DI_UnloadClampOpened");
       #sUPS_Fault(iHWStatus := "DI_UPS_Fault");
       #sInternalGateLocked(iHWStatus := NOT "DI_InternalGateLocked");
       #sExternalGateLocked(iHWStatus := NOT "DI_ExternalGateLocked");
       #sInverterActive(iHWStatus := "DI_InverterActive");
       #sUnloadClampNotClosedWithPart(iHWStatus := "DI_UnloadClampNotClosedWithPart");
       //
       #sFreeI5_0(iHWStatus := "DI_FreeI5_0");
       #sFreeI5_1(iHWStatus := "DI_FreeI5_1");
       #sInternalGateOpened(iHWStatus := "DI_InternalGateOpened");
       #sExternalGateOpened(iHWStatus := "DI_ExternalGateOpened");
       #sPowerMeterBackCtrl(iHWStatus := "DI_PowerMeterBackCtrl");
       #sPowerMeterFrontCtrl(iHWStatus := "DI_PowerMeterFrontCtrl");
       #sFreeI5_6(iHWStatus := "DI_FreeI5_6");
       #sFreeI5_7(iHWStatus := "DI_FreeI5_7");
   END_REGION

   REGION I6.0 - I7.7 : DI 16x24VDC ST Slot 4
       #sHeadChillerCutOff(iHWStatus := "DI_HeadChillerCutOff");
       #sHeadChillerTemperature(iHWStatus := "DI_HeadChillerTemperature");
       #sFreeI6_2(iHWStatus := "DI_FreeI6_2");
       #sFreeI6_3(iHWStatus := "DI_FreeI6_3");
       #sClampingOpenCtrl(iHWStatus := "DI_ClampingOpenCtrl");
       #sB_Axis_BrakeReleasedCtrl(iHWStatus := "DI_B_AxisBrakeReleasedCtrl");
       #sFreeI6_6(iHWStatus := "DI_FreeI6.6");
       #sB_AxisReferencePoint(iHWStatus := "DI_B_AxisReferencePoint");
       //
       #sSourceChillerHighPressure(iHWStatus := "DI_SourceChillerHighPressure");
       #sSourceChillerWaterTemperature(iHWStatus := "DI_SourceChillerWaterTemperature");
       #sSourceChillerFlow(iHWStatus := "DI_SourceChillerFlow");
       #sSourceChillerCollectivFault(iHWStatus := "DI_SourceChillerCollectivFault");
       #sSourceChillerWaterLevel(iHWStatus := "DI_SourceChillerWaterLevel");
       #sSourceChillerAmbiantTemperature(iHWStatus := "DI_SourceChillerAmbiantTemperature");
       #sSourceChillerCutOff(iHWStatus := "DI_SourceChillerCutOff");
       #sSourceChillerTemperature(iHWStatus := "DI_SourceChillerTemperature");
   END_REGION
END_FUNCTION_BLOCK

FUNCTION_BLOCK "FB_DigitalInput"   // FB15, SCL
{ S7_Optimized_Access := 'TRUE' }
// stored: AutoNumber false, MemoryReserve 100, SetENOAutomatically false
   VAR_INPUT
      iHWStatus { ExternalAccessible := 'False'; ExternalVisible := 'False'; ExternalWritable := 'False'} : Bool;   // PLC Digital Input Hardware status
   END_VAR
   VAR
      sDBI_F_Trig { S7_SetPoint := 'True'} : F_TRIG;
      sDBI_R_Trig { S7_SetPoint := 'True'} : R_TRIG;
      sSWStatus { ExternalAccessible := 'False'; ExternalVisible := 'False'; ExternalWritable := 'False'} : Bool;
      sSWPositiveFront { ExternalAccessible := 'False'; ExternalVisible := 'False'; ExternalWritable := 'False'} : Bool;
      sSWNegativeFront { ExternalAccessible := 'False'; ExternalVisible := 'False'; ExternalWritable := 'False'} : Bool;
   END_VAR
BEGIN
   REGION Description header 
       //==================================================================================
       // POSALUX Swiss SA / (C) Copyright 2024
       //----------------------------------------------------------------------------------
       // Title: Fonction Digital Input
       // Comment/Function: This function handles the state of a digital input, including
       //                   edge detection. It reads the hardware state, updates the
       //                   software state, and detects rising and falling edges.
       // Author: Gowsigan SRITHARAN
       // Engineering: TIA Portal v17
       //----------------------------------------------------------------------------------
       // Change log table:
       // Version  | Date     | Expert in charge | Changes applied
       // ---------|----------|------------------|-----------------------------------------
       // 00.00.01 | 20250106 | GSR              | First released version
       // =================================================================================
   END_REGION

   REGION Mise à jour de l'état de l'entree
       #sSWStatus:= #iHWStatus;
   END_REGION

   REGION Détection des fronts
       #sDBI_R_Trig(CLK := #sSWStatus,
                   Q => #sSWPositiveFront);

       #sDBI_F_Trig(CLK:=#sSWStatus,
                   Q=>#sSWNegativeFront);
   END_REGION
END_FUNCTION_BLOCK

FUNCTION_BLOCK "FB_DigitalInputsSonplas"   // FB211, SCL
{ S7_Optimized_Access := 'TRUE' }
// stored: AutoNumber false, MemoryReserve 100, SetENOAutomatically false
   VAR
      sSonplasDiagDPCoupler { S7_SetPoint := 'True'} : "FB_DigitalInput";
      sSonplasReady { S7_SetPoint := 'True'} : "FB_DigitalInput";
      sSonplasNoEStop { S7_SetPoint := 'True'} : "FB_DigitalInput";
      sSonplasDoorsClosed { S7_SetPoint := 'True'} : "FB_DigitalInput";
      sSonplasRunError { S7_SetPoint := 'True'} : "FB_DigitalInput";
      sSonplasFreeI200_5 { S7_SetPoint := 'True'} : "FB_DigitalInput";
      sSonplasFreeI200_6 { S7_SetPoint := 'True'} : "FB_DigitalInput";
      sSonplasFreeI200_7 { S7_SetPoint := 'True'} : "FB_DigitalInput";
      sSonplasFreeI201_0 { S7_SetPoint := 'True'} : "FB_DigitalInput";
      sSonplasOutCollision { S7_SetPoint := 'True'} : "FB_DigitalInput";
      sSonplasFreeI201_2 { S7_SetPoint := 'True'} : "FB_DigitalInput";
      Sonpla_FreeI201_3 { S7_SetPoint := 'True'} : "FB_DigitalInput";
      sSonplasFreeI201_4 { S7_SetPoint := 'True'} : "FB_DigitalInput";
      sSonplasFreeI201_5 { S7_SetPoint := 'True'} : "FB_DigitalInput";
      sSonplasFreeI201_6 { S7_SetPoint := 'True'} : "FB_DigitalInput";
      sSonplasFreeI201_7 { S7_SetPoint := 'True'} : "FB_DigitalInput";
      sSonplasShuttle1Finished { S7_SetPoint := 'True'} : "FB_DigitalInput";
      sSonplasFreeI202_1 { S7_SetPoint := 'True'} : "FB_DigitalInput";
      sSonplasFreeI202_2 { S7_SetPoint := 'True'} : "FB_DigitalInput";
      sSonplasFreeI202_3 { S7_SetPoint := 'True'} : "FB_DigitalInput";
      sSonplasFreeI202_4 { S7_SetPoint := 'True'} : "FB_DigitalInput";
      sSonplasFreeI202_5 { S7_SetPoint := 'True'} : "FB_DigitalInput";
      sSonplasFreeI202_6 { S7_SetPoint := 'True'} : "FB_DigitalInput";
      sSonplasFreeI202_7 { S7_SetPoint := 'True'} : "FB_DigitalInput";
      sSonplasShuttle2Finished { S7_SetPoint := 'True'} : "FB_DigitalInput";
      sSonplasFreeI203_1 { S7_SetPoint := 'True'} : "FB_DigitalInput";
      sSonplasFreeI203_2 { S7_SetPoint := 'True'} : "FB_DigitalInput";
      sSonplasFreeI203_3 { S7_SetPoint := 'True'} : "FB_DigitalInput";
      sSonplasFreeI203_4 { S7_SetPoint := 'True'} : "FB_DigitalInput";
      sSonplasFreeI203_5 { S7_SetPoint := 'True'} : "FB_DigitalInput";
      sSonplasFreeI203_6 { S7_SetPoint := 'True'} : "FB_DigitalInput";
      sSonplasFreeI203_7 { S7_SetPoint := 'True'} : "FB_DigitalInput";
      sSonplasFlowResultAvail { S7_SetPoint := 'True'} : "FB_DigitalInput";
      sSonplasFreeI244_1 { S7_SetPoint := 'True'} : "FB_DigitalInput";
      sSonplasFreeI244_2 { S7_SetPoint := 'True'} : "FB_DigitalInput";
      sSonplasFreeI244_3 { S7_SetPoint := 'True'} : "FB_DigitalInput";
      sSonplasFreeI244_4 { S7_SetPoint := 'True'} : "FB_DigitalInput";
      sSonplasFreeI244_5 { S7_SetPoint := 'True'} : "FB_DigitalInput";
      sSonplasFreeI244_6 { S7_SetPoint := 'True'} : "FB_DigitalInput";
      sSonplasFreeI244_7 { S7_SetPoint := 'True'} : "FB_DigitalInput";
   END_VAR
BEGIN
   REGION Description head
       //==================================================================================
       // POSALUX Swiss SA / (C) Copyright 2025
       //----------------------------------------------------------------------------------
       // Title: Digital Inputs mapping
       // Comment/Function: Sonplas Digital Inputs mapping
       // Author: Fabien WALDT
       // Engineering: TIA Portal v17
       //----------------------------------------------------------------------------------
       // Change log table:
       // Version  | Date     | Expert in charge | Changes applied
       // ---------|----------|------------------|-----------------------------------------
       // 00.00.01 | 20250423 | WFA              | First released version
       // =================================================================================
   END_REGION


   REGION Operating modes and parts exchange
       #sSonplasDiagDPCoupler(iHWStatus := "DI_SonplasDiagDPCoupler");
       #sSonplasReady(iHWStatus := "DI_SonplasReady");
       #sSonplasNoEStop(iHWStatus := "DI_SonplasNoEStop");
       #sSonplasDoorsClosed(iHWStatus := "DI_SonplasDoorsClosed");
       #sSonplasRunError(iHWStatus := "DI_SonplasRunError");
       #sSonplasFreeI200_5(iHWStatus := "DI_SonplasFreeI200_5");
       #sSonplasFreeI200_6(iHWStatus := "DI_SonplasFreeI200_6");
       #sSonplasFreeI200_7(iHWStatus := "DI_SonplasFreeI200_7");
       // 
       #sSonplasFreeI201_0(iHWStatus := "DI_SonplasFreeI201_0");
       #sSonplasOutCollision(iHWStatus := "DI_SonplasOutCollision");
       #sSonplasFreeI201_2(iHWStatus := "DI_SonplasFreeI201_2");
       #Sonpla_FreeI201_3(iHWStatus := "DI_SonplasFreeI201_3");
       #sSonplasFreeI201_4(iHWStatus := "DI_SonplasFreeI201_4");
       #sSonplasFreeI201_5(iHWStatus := "DI_SonplasFreeI201_5");
       #sSonplasFreeI201_6(iHWStatus := "DI_SonplasFreeI201_6");
       #sSonplasFreeI201_7(iHWStatus := "DI_SonplasFreeI201_7");
   END_REGION

   REGION Part exchange
       #sSonplasShuttle1Finished(iHWStatus := "DI_SonplasShuttle1Finished");
       #sSonplasFreeI202_1(iHWStatus := "DI_SonplasFreeI202_1");
       #sSonplasFreeI202_2(iHWStatus := "DI_SonplasFreeI202_2");
       #sSonplasFreeI202_3(iHWStatus := "DI_SonplasFreeI202_3");
       #sSonplasFreeI202_4(iHWStatus := "DI_SonplasFreeI202_4");
       #sSonplasFreeI202_5(iHWStatus := "DI_SonplasFreeI202_5");
       #sSonplasFreeI202_6(iHWStatus := "DI_SonplasFreeI202_6");
       #sSonplasFreeI202_7(iHWStatus := "DI_SonplasFreeI202_7");
       //
       #sSonplasShuttle2Finished(iHWStatus := "DI_SonplasShuttle2Finished");
       #sSonplasFreeI203_1(iHWStatus := "DI_SonplasFreeI203_1");
       #sSonplasFreeI203_2(iHWStatus := "DI_SonplasFreeI203_2");
       #sSonplasFreeI203_3(iHWStatus := "DI_SonplasFreeI203_3");
       #sSonplasFreeI203_4(iHWStatus := "DI_SonplasFreeI203_4");
       #sSonplasFreeI203_5(iHWStatus := "DI_SonplasFreeI203_5");
       #sSonplasFreeI203_6(iHWStatus := "DI_SonplasFreeI203_6");
       #sSonplasFreeI203_7(iHWStatus := "DI_SonplasFreeI203_7");
   END_REGION

   REGION Measure
       #sSonplasFlowResultAvail(iHWStatus := "DI_SonplasFlowResultAvail");
       #sSonplasFreeI244_1(iHWStatus := "DI_SonplasFreeI244_1");
       #sSonplasFreeI244_2(iHWStatus := "DI_SonplasFreeI244_2");
       #sSonplasFreeI244_3(iHWStatus := "DI_SonplasFreeI244_3");
       #sSonplasFreeI244_4(iHWStatus := "DI_SonplasFreeI244_4");
       #sSonplasFreeI244_5(iHWStatus := "DI_SonplasFreeI244_5");
       #sSonplasFreeI244_6(iHWStatus := "DI_SonplasFreeI244_6");
       #sSonplasFreeI244_7(iHWStatus := "DI_SonplasFreeI244_7");
   END_REGION
END_FUNCTION_BLOCK

FUNCTION_BLOCK "FB_DigitalInputsBW_Station"   // FB214, SCL
{ S7_Optimized_Access := 'TRUE' }
// stored: AutoNumber false, MemoryReserve 100, SetENOAutomatically false
   VAR
      sUndrilledPartCtrl { S7_SetPoint := 'True'} : "FB_DigitalInput";
      sDrilledPartCtrl { S7_SetPoint := 'True'} : "FB_DigitalInput";
      sBwCtrl { S7_SetPoint := 'True'} : "FB_DigitalInput";
   END_VAR
BEGIN
   REGION Description head
       //==================================================================================
       // POSALUX Swiss SA / (C) Copyright 2025
       //----------------------------------------------------------------------------------
       // Title: Digital Inputs mapping
       // Comment/Function: BW Station Digital Inputs mapping
       // Author: Fabien WALDT
       // Engineering: TIA Portal v17
       //----------------------------------------------------------------------------------
       // Change log table:
       // Version  | Date     | Expert in charge | Changes applied
       // ---------|----------|------------------|-----------------------------------------
       // 00.00.01 | 20250423 | WFA              | First released version
       // =================================================================================
   END_REGION


   REGION Backwall Station 
       IF "DB_WAF".CtrlInEnable OR "DB_WAF".CtrlOutEnable THEN
           #sUndrilledPartCtrl(iHWStatus := "DB_BwLoaderExchange".Inputs.UndrilledPartControl);
       END_IF;
       IF "DB_WAF".CtrlInEnable OR "DB_WAF".CtrlOutEnable THEN
           #sDrilledPartCtrl(iHWStatus := "DB_BwLoaderExchange".Inputs.DrilledPartControl);
       END_IF;
       IF "DB_WAF".CtrlBwEnable THEN
           #sBwCtrl(iHWStatus := "DB_BwLoaderExchange".Inputs.BackwallControl);
       END_IF;
   END_REGION
END_FUNCTION_BLOCK

FUNCTION_BLOCK "FB_AnalogOutputs"   // FB225, SCL
{ S7_Optimized_Access := 'TRUE' }
// stored: AutoNumber false, MemoryReserve 100, SetENOAutomatically false
   VAR
      sNozzleOverpressureSetPoint { S7_SetPoint := 'True'} : "FB_AnalogOutput";
      sFreeQW482 { S7_SetPoint := 'True'} : "FB_AnalogOutput";
      sVentilatorSetPoint { S7_SetPoint := 'True'} : "FB_AnalogOutput";
      sPropValveClimSetPoint { S7_SetPoint := 'True'} : "FB_AnalogOutput";
   END_VAR
BEGIN
   REGION Description head
       //==================================================================================
       // POSALUX Swiss SA / (C) Copyright 2025
       //----------------------------------------------------------------------------------
       // Title: Analog output function
       // Comment/Function: Analog Ouputs mapping
       // Author: Fabien WALDT
       // Engineering: TIA Portal v17
       //----------------------------------------------------------------------------------
       // Change log table:
       // Version  | Date     | Expert in charge | Changes applied
       // ---------|----------|------------------|-----------------------------------------
       // 00.00.01 | 20250423 | WFA              | First released version
       // =================================================================================
   END_REGION

   // ET200SP Mapping
   REGION IW428 - IW434 : AQ 4xU/I ST Slot 22
       #sNozzleOverpressureSetPoint(iLimitUp := 10.0,
                                    iLimitDown := 0.0,
                                    iMaxAIWordValue := 27648.0,
                                    oValueHW => "AQ_NozzleOverpressureSetPoint");

       #sFreeQW482(iLimitUp := 100.0,
                   iLimitDown := 0.0,
                   iMaxAIWordValue := 27648.0,
                   oValueHW => "AQ_FreeQW482");

       #sVentilatorSetPoint(iLimitUp := 100.0,
                            iLimitDown := 0.0,
                            iMaxAIWordValue := 27648.0,
                            oValueHW => "AQ_VentilatorSetPoint");

       #sPropValveClimSetPoint(iLimitUp := 100.0,
                               iLimitDown := 0.0,
                               iMaxAIWordValue := 27648.0,
                               oValueHW => "AQ_PropValveClimSetPoint");
   END_REGION
END_FUNCTION_BLOCK

FUNCTION_BLOCK "FB_AnalogOutput"   // FB33, SCL
{ S7_Optimized_Access := 'TRUE' }
// stored: AutoNumber false, MemoryReserve 100, SetENOAutomatically false
   VAR_INPUT
      iLimitUp { ExternalAccessible := 'False'; ExternalVisible := 'False'; ExternalWritable := 'False'} : Real;   // Limit up real value
      iLimitDown { ExternalAccessible := 'False'; ExternalVisible := 'False'; ExternalWritable := 'False'} : Real;   // Limit down real value
      iMaxAIWordValue { ExternalAccessible := 'False'; ExternalVisible := 'False'; ExternalWritable := 'False'} : Real;   // Word analog output range
   END_VAR
   VAR_OUTPUT
      oValueHW { ExternalAccessible := 'False'; ExternalVisible := 'False'; ExternalWritable := 'False'} : Word;   // Value in word for PLC analog output
   END_VAR
   VAR
      sSWRealValue { ExternalAccessible := 'False'; ExternalVisible := 'False'; ExternalWritable := 'False'} : Real;
      sHWWordValue { ExternalAccessible := 'False'; ExternalVisible := 'False'; ExternalWritable := 'False'} : Word;
   END_VAR
   VAR_TEMP
      tValueSWInt : Int;   // Int value (conversion)
      tValueSWWord : Word;   // Word value to set as PLC analog output
      tRange : Real;   // Real value range
      tValueSWReal : Real;   // Real value in absolute
   END_VAR
BEGIN
   REGION Description header 
       //==================================================================================
       // POSALUX Swiss SA / (C) Copyright 2024
       //----------------------------------------------------------------------------------
       // Title: Analog output function
       // Comment/Function: This function handles analog value conversion AND scaling.  
       //                   It converts a real value to an integer value, then to a word
       //                   for the PLC's analog output. The function also performs scaling
       //                   based on specified limits.
       // Author: Gowsigan SRITHARAN
       // Engineering: TIA Portal v17
       //----------------------------------------------------------------------------------
       // Change log table:
       // Version  | Date     | Expert in charge | Changes applied
       // ---------|----------|------------------|-----------------------------------------
       // 00.00.01 | 20250106 | GSR              | First released version
       // =================================================================================
   END_REGION

   REGION Initialization
       #tValueSWReal := #sSWRealValue;
   END_REGION

   REGION Absolute Value Calculation and Scaling
       // Calculate range
       #tRange := #iLimitUp - #iLimitDown;

       // Scale the value
       #tValueSWReal := #tValueSWReal - #iLimitDown;
       #tValueSWReal := #tValueSWReal / #tRange;
       #tValueSWReal := #tValueSWReal * #iMaxAIWordValue;
   END_REGION

   REGION Real-to-Word Value Conversion
       // Convert REAL to INT
       #tValueSWInt := REAL_TO_INT(#tValueSWReal);

       // Convert INT to WORD
       #tValueSWWord := INT_TO_WORD(#tValueSWInt);

       // Assign output values
       #sHWWordValue := #tValueSWWord;
       #oValueHW := #tValueSWWord;
   END_REGION
END_FUNCTION_BLOCK

